// TwinCAT 3 PLC project DMMS_PLC
// ProgramVersion: 3.1.4026.19
// libraries:
//   Tc2_Standard, * (Beckhoff Automation GmbH)
//   Tc2_System, * (Beckhoff Automation GmbH)
//   Tc3_Mc3PlanarMotion, * (Beckhoff Automation GmbH)
//   Tc3_Physics, * (Beckhoff Automation GmbH)
//   Tc3_XPlanarStandard, * (Beckhoff Automation GmbH)
//   Tc3_XPlanarUtility, * (Beckhoff Automation GmbH)
// project tree:
//   DUTs/Communiction/GlobalStatus/ ST_ComIn_GlobalStatus.TcDUT (not stored), ST_ComOut_GlobalStatus.TcDUT (not stored), ST_Com_GlobalStatus.TcDUT (not stored)
//   DUTs/Communiction/Movers/ ST_ComIn_ExportMover.TcDUT (not stored), ST_ComOut_ExportMover.TcDUT, ST_Com_ExportMover.TcDUT (not stored)
//   DUTs/Communiction/Station/ ST_ComIn_ExportStation.TcDUT (not stored), ST_ComOut_ExportStation.TcDUT (not stored), ST_Com_ExportStation.TcDUT
//   GVLs/ Communication.TcGVL (not stored), Debug.TcGVL (not stored), GVL.TcGVL (not stored)
//   Mover/DUTs/ MoverPositionUnion.TcDUT, ST_ControlData.TcDUT (not stored), ST_EMoverLoadType.TcDUT (not stored), ST_ManMov_FreeMove.TcDUT, ST_ManMov_MoveTrack.TcDUT (not stored), ST_ManualMovements.TcDUT (not stored), ST_MoverConfiguration.TcDUT (not stored), ST_ProcessResult.TcDUT, ST_ProcessTask.TcDUT (not stored), ST_ProductData.TcDUT (not stored), ST_WellplateParametrization.TcDUT (not stored)
//   Mover/ FB_ApplicationMover.TcPOU, I_MoverApplication.TcIO
//   / PlcTask.TcTTO
//   POUs/ FB_MotionSystem.TcPOU, MAIN.TcPOU (not stored)
//   Stations/Base/ FB_StationBase.TcPOU, I_Station.TcIO
//   Stations/DUTs/ E_ProcessMode.TcDUT (not stored), ST_EStationProcessState.TcDUT (not stored), ST_EStationHandshake.TcDUT (not stored), ST_StationPosition.TcDUT (not stored), ST_StationReturn.TcDUT, ST_VisStationData.TcDUT (not stored)
//   Stations/ FB_PuncherStation.TcPOU (not stored), FB_PuncherSeparateStation.TcPOU, FB_PuncherBufferStation.TcPOU
//   Stations/Helper/ FB_HistoryInfo.TcPOU
//   Tracks/Base/ FB_BaseTrack.TcPOU (not stored), I_Track.TcIO (not stored)
//   Tracks/ FB_CloseLoopTrack.TcPOU (not stored), FB_UserInteractionTrack.TcPOU (not stored), FB_PipettePreBufferTrack.TcPOU (not stored), FB_PipetteTrack.TcPOU (not stored), FB_PipettePostBufferTrack.TcPOU, FB_PipetteBufferConTrack.TcPOU (not stored), FB_PuncherWellplateTrack.TcPOU, FB_PuncherBufferTrack.TcPOU (not stored), FB_StradeFirstSegTrack.TcPOU, FB_StradeSecondSegTrack.TcPOU (not stored), FB_PuncherSeperateTrack.TcPOU (not stored)
// real-time tasks:
//   TASK Job Task: cycle default, priority 2
//   TASK MC-Task (MET): cycle T#2ms, priority 3, ADS port 351
//   TASK MC-Task (MPT): cycle T#10ms, priority 4, ADS port 352
//   TASK PlcTask: cycle T#10ms, priority 20, ADS port 353
//   TASK XPlanar Task_0: cycle T#250us, priority 1, ADS port 350
//   TASK XPlanar Task_10: cycle T#250us, priority 5, ADS port 354
// I/O:
//   DEVICE Device 2 (EtherCAT), AmsNetId 192.168.2.44.3.1
//     Term 1 (APS4322-7000) [APS4322-7000 Drive]
//       Term 2 (APS4322-5000) [APS4322-5000 Feedback]
//     Term 3 (APS4322-7000) [APS4322-7000 Drive]
//       Term 4 (APS4322-5000) [APS4322-5000 Feedback]
//     Term 5 (APS4322-7000) [APS4322-7000 Drive]
//       Term 6 (APS4322-5000) [APS4322-5000 Feedback]
//     Term 7 (APS4322-7000) [APS4322-7000 Drive]
//       Term 8 (APS4322-5000) [APS4322-5000 Feedback]
//     Term 9 (APS4322-7000) [APS4322-7000 Drive]
//       Term 10 (APS4322-5000) [APS4322-5000 Feedback]
// variable links:
//   Device 2 (EtherCAT) <-> TcCOM Objects/XPlanar/Part1/APS4322_P1_1
//     Term 1 (APS4322-7000)/APS Comm Inputs/CommStatusWord <-> Data Pointer/MoverCommStatusWord
//     Term 1 (APS4322-7000)/APS Comm Inputs/Data {1..4} <-> Data Pointer/MoverCommDataIn[{0..3}]  (4 links)
//     Term 1 (APS4322-7000)/APS Comm Outputs/CommControlWord <-> Data Pointer/MoverCommControlWord
//     Term 1 (APS4322-7000)/APS Comm Outputs/Data 1 <-> Data Pointer/MoverCommDataOut
//     Term 1 (APS4322-7000)/APS Diagdata/DC Link Voltage <-> Data Pointer/DcLinkVoltage
//     Term 1 (APS4322-7000)/APS Diagdata/Power supply current <-> Data Pointer/PowerSupplyCurrent
//     Term 1 (APS4322-7000)/APS Inputs/StatusWord <-> Data Pointer/PowerUnitStatusWord
//     Term 1 (APS4322-7000)/APS Outputs/ControlWord <-> Data Pointer/PowerUnitControlWord
//     Term 1 (APS4322-7000)/APS Outputs/Current D 0X0 <-> Data Pointer/DCurrentSetPoints[0]
//     Term 1 (APS4322-7000)/APS Outputs/Current D 0X1 <-> Data Pointer/DCurrentSetPoints[1]
//     Term 1 (APS4322-7000)/APS Outputs/Current D 0X2 <-> Data Pointer/DCurrentSetPoints[2]
//     Term 1 (APS4322-7000)/APS Outputs/Current D 1X0 <-> Data Pointer/DCurrentSetPoints[6]
//     Term 1 (APS4322-7000)/APS Outputs/Current D 1X1 <-> Data Pointer/DCurrentSetPoints[7]
//     Term 1 (APS4322-7000)/APS Outputs/Current D 1X2 <-> Data Pointer/DCurrentSetPoints[8]
//     Term 1 (APS4322-7000)/APS Outputs/Current D 2X0 <-> Data Pointer/DCurrentSetPoints[12]
//     Term 1 (APS4322-7000)/APS Outputs/Current D 2X1 <-> Data Pointer/DCurrentSetPoints[13]
//     Term 1 (APS4322-7000)/APS Outputs/Current D 2X2 <-> Data Pointer/DCurrentSetPoints[14]
//     Term 1 (APS4322-7000)/APS Outputs/Current D 3X0 <-> Data Pointer/DCurrentSetPoints[18]
//     Term 1 (APS4322-7000)/APS Outputs/Current D 3X1 <-> Data Pointer/DCurrentSetPoints[19]
//     Term 1 (APS4322-7000)/APS Outputs/Current D 3X2 <-> Data Pointer/DCurrentSetPoints[20]
//     Term 1 (APS4322-7000)/APS Outputs/Current D 0Y0 <-> Data Pointer/DCurrentSetPoints[3]
//     Term 1 (APS4322-7000)/APS Outputs/Current D 0Y1 <-> Data Pointer/DCurrentSetPoints[4]
//     Term 1 (APS4322-7000)/APS Outputs/Current D 0Y2 <-> Data Pointer/DCurrentSetPoints[5]
//     Term 1 (APS4322-7000)/APS Outputs/Current D 1Y0 <-> Data Pointer/DCurrentSetPoints[9]
//     Term 1 (APS4322-7000)/APS Outputs/Current D 1Y1 <-> Data Pointer/DCurrentSetPoints[10]
//     Term 1 (APS4322-7000)/APS Outputs/Current D 1Y2 <-> Data Pointer/DCurrentSetPoints[11]
//     Term 1 (APS4322-7000)/APS Outputs/Current D 2Y0 <-> Data Pointer/DCurrentSetPoints[15]
//     Term 1 (APS4322-7000)/APS Outputs/Current D 2Y1 <-> Data Pointer/DCurrentSetPoints[16]
//     Term 1 (APS4322-7000)/APS Outputs/Current D 2Y2 <-> Data Pointer/DCurrentSetPoints[17]
//     Term 1 (APS4322-7000)/APS Outputs/Current D 3Y0 <-> Data Pointer/DCurrentSetPoints[21]
//     Term 1 (APS4322-7000)/APS Outputs/Current D 3Y1 <-> Data Pointer/DCurrentSetPoints[22]
//     Term 1 (APS4322-7000)/APS Outputs/Current D 3Y2 <-> Data Pointer/DCurrentSetPoints[23]
//     Term 1 (APS4322-7000)/APS Outputs/Current Q 0X0 <-> Data Pointer/QCurrentSetPoints[0]
//     Term 1 (APS4322-7000)/APS Outputs/Current Q 0X1 <-> Data Pointer/QCurrentSetPoints[1]
//     Term 1 (APS4322-7000)/APS Outputs/Current Q 0X2 <-> Data Pointer/QCurrentSetPoints[2]
//     Term 1 (APS4322-7000)/APS Outputs/Current Q 1X0 <-> Data Pointer/QCurrentSetPoints[6]
//     Term 1 (APS4322-7000)/APS Outputs/Current Q 1X1 <-> Data Pointer/QCurrentSetPoints[7]
//     Term 1 (APS4322-7000)/APS Outputs/Current Q 1X2 <-> Data Pointer/QCurrentSetPoints[8]
//     Term 1 (APS4322-7000)/APS Outputs/Current Q 2X0 <-> Data Pointer/QCurrentSetPoints[12]
//     Term 1 (APS4322-7000)/APS Outputs/Current Q 2X1 <-> Data Pointer/QCurrentSetPoints[13]
//     Term 1 (APS4322-7000)/APS Outputs/Current Q 2X2 <-> Data Pointer/QCurrentSetPoints[14]
//     Term 1 (APS4322-7000)/APS Outputs/Current Q 3X0 <-> Data Pointer/QCurrentSetPoints[18]
//     Term 1 (APS4322-7000)/APS Outputs/Current Q 3X1 <-> Data Pointer/QCurrentSetPoints[19]
//     Term 1 (APS4322-7000)/APS Outputs/Current Q 3X2 <-> Data Pointer/QCurrentSetPoints[20]
//     Term 1 (APS4322-7000)/APS Outputs/Current Q 0Y0 <-> Data Pointer/QCurrentSetPoints[3]
//     Term 1 (APS4322-7000)/APS Outputs/Current Q 0Y1 <-> Data Pointer/QCurrentSetPoints[4]
//     Term 1 (APS4322-7000)/APS Outputs/Current Q 0Y2 <-> Data Pointer/QCurrentSetPoints[5]
//     Term 1 (APS4322-7000)/APS Outputs/Current Q 1Y0 <-> Data Pointer/QCurrentSetPoints[9]
//     Term 1 (APS4322-7000)/APS Outputs/Current Q 1Y1 <-> Data Pointer/QCurrentSetPoints[10]
//     Term 1 (APS4322-7000)/APS Outputs/Current Q 1Y2 <-> Data Pointer/QCurrentSetPoints[11]
//     Term 1 (APS4322-7000)/APS Outputs/Current Q 2Y0 <-> Data Pointer/QCurrentSetPoints[15]
//     Term 1 (APS4322-7000)/APS Outputs/Current Q 2Y1 <-> Data Pointer/QCurrentSetPoints[16]
//     Term 1 (APS4322-7000)/APS Outputs/Current Q 2Y2 <-> Data Pointer/QCurrentSetPoints[17]
//     Term 1 (APS4322-7000)/APS Outputs/Current Q 3Y0 <-> Data Pointer/QCurrentSetPoints[21]
//     Term 1 (APS4322-7000)/APS Outputs/Current Q 3Y1 <-> Data Pointer/QCurrentSetPoints[22]
//     Term 1 (APS4322-7000)/APS Outputs/Current Q 3Y2 <-> Data Pointer/QCurrentSetPoints[23]
//     Term 1 (APS4322-7000)/APS Outputs/PhiE 0X0 <-> Data Pointer/PhiSetPoints[0]
//     Term 1 (APS4322-7000)/APS Outputs/PhiE 0X1 <-> Data Pointer/PhiSetPoints[1]
//     Term 1 (APS4322-7000)/APS Outputs/PhiE 0X2 <-> Data Pointer/PhiSetPoints[2]
//     Term 1 (APS4322-7000)/APS Outputs/PhiE 1X0 <-> Data Pointer/PhiSetPoints[6]
//     Term 1 (APS4322-7000)/APS Outputs/PhiE 1X1 <-> Data Pointer/PhiSetPoints[7]
//     Term 1 (APS4322-7000)/APS Outputs/PhiE 1X2 <-> Data Pointer/PhiSetPoints[8]
//     Term 1 (APS4322-7000)/APS Outputs/PhiE 2X0 <-> Data Pointer/PhiSetPoints[12]
//     Term 1 (APS4322-7000)/APS Outputs/PhiE 2X1 <-> Data Pointer/PhiSetPoints[13]
//     Term 1 (APS4322-7000)/APS Outputs/PhiE 2X2 <-> Data Pointer/PhiSetPoints[14]
//     Term 1 (APS4322-7000)/APS Outputs/PhiE 3X0 <-> Data Pointer/PhiSetPoints[18]
//     Term 1 (APS4322-7000)/APS Outputs/PhiE 3X1 <-> Data Pointer/PhiSetPoints[19]
//     Term 1 (APS4322-7000)/APS Outputs/PhiE 3X2 <-> Data Pointer/PhiSetPoints[20]
//     Term 1 (APS4322-7000)/APS Outputs/PhiE 0Y0 <-> Data Pointer/PhiSetPoints[3]
//     Term 1 (APS4322-7000)/APS Outputs/PhiE 0Y1 <-> Data Pointer/PhiSetPoints[4]
//     Term 1 (APS4322-7000)/APS Outputs/PhiE 0Y2 <-> Data Pointer/PhiSetPoints[5]
//     Term 1 (APS4322-7000)/APS Outputs/PhiE 1Y0 <-> Data Pointer/PhiSetPoints[9]
//     Term 1 (APS4322-7000)/APS Outputs/PhiE 1Y1 <-> Data Pointer/PhiSetPoints[10]
//     Term 1 (APS4322-7000)/APS Outputs/PhiE 1Y2 <-> Data Pointer/PhiSetPoints[11]
//     Term 1 (APS4322-7000)/APS Outputs/PhiE 2Y0 <-> Data Pointer/PhiSetPoints[15]
//     Term 1 (APS4322-7000)/APS Outputs/PhiE 2Y1 <-> Data Pointer/PhiSetPoints[16]
//     Term 1 (APS4322-7000)/APS Outputs/PhiE 2Y2 <-> Data Pointer/PhiSetPoints[17]
//     Term 1 (APS4322-7000)/APS Outputs/PhiE 3Y0 <-> Data Pointer/PhiSetPoints[21]
//     Term 1 (APS4322-7000)/APS Outputs/PhiE 3Y1 <-> Data Pointer/PhiSetPoints[22]
//     Term 1 (APS4322-7000)/APS Outputs/PhiE 3Y2 <-> Data Pointer/PhiSetPoints[23]
//     Term 1 (APS4322-7000)/Term 2 (APS4322-5000)/FB Inputs/A{0..8 step 2} X-Field <-> Data Pointer/HallSensorFieldsXYZ[{0..12 step 3}]  (5 links)
//     Term 1 (APS4322-7000)/Term 2 (APS4322-5000)/FB Inputs/A{0..8 step 2} Y-Field <-> Data Pointer/HallSensorFieldsXYZ[{1..13 step 3}]  (5 links)
//     Term 1 (APS4322-7000)/Term 2 (APS4322-5000)/FB Inputs/A{0..8 step 2} Z-Field <-> Data Pointer/HallSensorFieldsXYZ[{2..14 step 3}]  (5 links)
//     Term 1 (APS4322-7000)/Term 2 (APS4322-5000)/FB Inputs/B{1..9 step 2} X-Field <-> Data Pointer/HallSensorFieldsXYZ[{15..27 step 3}]  (5 links)
//     Term 1 (APS4322-7000)/Term 2 (APS4322-5000)/FB Inputs/B{1..9 step 2} Y-Field <-> Data Pointer/HallSensorFieldsXYZ[{16..28 step 3}]  (5 links)
//     Term 1 (APS4322-7000)/Term 2 (APS4322-5000)/FB Inputs/B{1..9 step 2} Z-Field <-> Data Pointer/HallSensorFieldsXYZ[{17..29 step 3}]  (5 links)
//     Term 1 (APS4322-7000)/Term 2 (APS4322-5000)/FB Inputs/C{0..8 step 2} X-Field <-> Data Pointer/HallSensorFieldsXYZ[{30..42 step 3}]  (5 links)
//     Term 1 (APS4322-7000)/Term 2 (APS4322-5000)/FB Inputs/C{0..8 step 2} Y-Field <-> Data Pointer/HallSensorFieldsXYZ[{31..43 step 3}]  (5 links)
//     Term 1 (APS4322-7000)/Term 2 (APS4322-5000)/FB Inputs/C{0..8 step 2} Z-Field <-> Data Pointer/HallSensorFieldsXYZ[{32..44 step 3}]  (5 links)
//     Term 1 (APS4322-7000)/Term 2 (APS4322-5000)/FB Inputs/D{1..9 step 2} X-Field <-> Data Pointer/HallSensorFieldsXYZ[{45..57 step 3}]  (5 links)
//     Term 1 (APS4322-7000)/Term 2 (APS4322-5000)/FB Inputs/D{1..9 step 2} Y-Field <-> Data Pointer/HallSensorFieldsXYZ[{46..58 step 3}]  (5 links)
//     Term 1 (APS4322-7000)/Term 2 (APS4322-5000)/FB Inputs/D{1..9 step 2} Z-Field <-> Data Pointer/HallSensorFieldsXYZ[{47..59 step 3}]  (5 links)
//     Term 1 (APS4322-7000)/Term 2 (APS4322-5000)/FB Inputs/E{0..8 step 2} X-Field <-> Data Pointer/HallSensorFieldsXYZ[{60..72 step 3}]  (5 links)
//     Term 1 (APS4322-7000)/Term 2 (APS4322-5000)/FB Inputs/E{0..8 step 2} Y-Field <-> Data Pointer/HallSensorFieldsXYZ[{61..73 step 3}]  (5 links)
//     Term 1 (APS4322-7000)/Term 2 (APS4322-5000)/FB Inputs/E{0..8 step 2} Z-Field <-> Data Pointer/HallSensorFieldsXYZ[{62..74 step 3}]  (5 links)
//     Term 1 (APS4322-7000)/Term 2 (APS4322-5000)/FB Inputs/F{1..9 step 2} X-Field <-> Data Pointer/HallSensorFieldsXYZ[{75..87 step 3}]  (5 links)
//     Term 1 (APS4322-7000)/Term 2 (APS4322-5000)/FB Inputs/F{1..9 step 2} Y-Field <-> Data Pointer/HallSensorFieldsXYZ[{76..88 step 3}]  (5 links)
//     Term 1 (APS4322-7000)/Term 2 (APS4322-5000)/FB Inputs/F{1..9 step 2} Z-Field <-> Data Pointer/HallSensorFieldsXYZ[{77..89 step 3}]  (5 links)
//     Term 1 (APS4322-7000)/Term 2 (APS4322-5000)/FB Inputs/G{0..8 step 2} X-Field <-> Data Pointer/HallSensorFieldsXYZ[{90..102 step 3}]  (5 links)
//     Term 1 (APS4322-7000)/Term 2 (APS4322-5000)/FB Inputs/G{0..8 step 2} Y-Field <-> Data Pointer/HallSensorFieldsXYZ[{91..103 step 3}]  (5 links)
//     Term 1 (APS4322-7000)/Term 2 (APS4322-5000)/FB Inputs/G{0..8 step 2} Z-Field <-> Data Pointer/HallSensorFieldsXYZ[{92..104 step 3}]  (5 links)
//     Term 1 (APS4322-7000)/Term 2 (APS4322-5000)/FB Inputs/H{1..9 step 2} X-Field <-> Data Pointer/HallSensorFieldsXYZ[{105..117 step 3}]  (5 links)
//     Term 1 (APS4322-7000)/Term 2 (APS4322-5000)/FB Inputs/H{1..9 step 2} Y-Field <-> Data Pointer/HallSensorFieldsXYZ[{106..118 step 3}]  (5 links)
//     Term 1 (APS4322-7000)/Term 2 (APS4322-5000)/FB Inputs/H{1..9 step 2} Z-Field <-> Data Pointer/HallSensorFieldsXYZ[{107..119 step 3}]  (5 links)
//     Term 1 (APS4322-7000)/Term 2 (APS4322-5000)/FB Inputs/I{0..8 step 2} X-Field <-> Data Pointer/HallSensorFieldsXYZ[{120..132 step 3}]  (5 links)
//     Term 1 (APS4322-7000)/Term 2 (APS4322-5000)/FB Inputs/I{0..8 step 2} Y-Field <-> Data Pointer/HallSensorFieldsXYZ[{121..133 step 3}]  (5 links)
//     Term 1 (APS4322-7000)/Term 2 (APS4322-5000)/FB Inputs/I{0..8 step 2} Z-Field <-> Data Pointer/HallSensorFieldsXYZ[{122..134 step 3}]  (5 links)
//     Term 1 (APS4322-7000)/Term 2 (APS4322-5000)/FB Inputs/J{1..9 step 2} X-Field <-> Data Pointer/HallSensorFieldsXYZ[{135..147 step 3}]  (5 links)
//     Term 1 (APS4322-7000)/Term 2 (APS4322-5000)/FB Inputs/J{1..9 step 2} Y-Field <-> Data Pointer/HallSensorFieldsXYZ[{136..148 step 3}]  (5 links)
//     Term 1 (APS4322-7000)/Term 2 (APS4322-5000)/FB Inputs/J{1..9 step 2} Z-Field <-> Data Pointer/HallSensorFieldsXYZ[{137..149 step 3}]  (5 links)
//     Term 1 (APS4322-7000)/Term 2 (APS4322-5000)/FB Inputs/Status <-> Data Pointer/FeedbackStatus
//   Device 2 (EtherCAT) <-> TcCOM Objects/XPlanar/Part1/APS4322_P1_2
//     Term 3 (APS4322-7000)/APS Comm Inputs/CommStatusWord <-> Data Pointer/MoverCommStatusWord
//     Term 3 (APS4322-7000)/APS Comm Inputs/Data {1..4} <-> Data Pointer/MoverCommDataIn[{0..3}]  (4 links)
//     Term 3 (APS4322-7000)/APS Comm Outputs/CommControlWord <-> Data Pointer/MoverCommControlWord
//     Term 3 (APS4322-7000)/APS Comm Outputs/Data 1 <-> Data Pointer/MoverCommDataOut
//     Term 3 (APS4322-7000)/APS Diagdata/DC Link Voltage <-> Data Pointer/DcLinkVoltage
//     Term 3 (APS4322-7000)/APS Diagdata/Power supply current <-> Data Pointer/PowerSupplyCurrent
//     Term 3 (APS4322-7000)/APS Inputs/StatusWord <-> Data Pointer/PowerUnitStatusWord
//     Term 3 (APS4322-7000)/APS Outputs/ControlWord <-> Data Pointer/PowerUnitControlWord
//     Term 3 (APS4322-7000)/APS Outputs/Current D 0X0 <-> Data Pointer/DCurrentSetPoints[0]
//     Term 3 (APS4322-7000)/APS Outputs/Current D 0X1 <-> Data Pointer/DCurrentSetPoints[1]
//     Term 3 (APS4322-7000)/APS Outputs/Current D 0X2 <-> Data Pointer/DCurrentSetPoints[2]
//     Term 3 (APS4322-7000)/APS Outputs/Current D 1X0 <-> Data Pointer/DCurrentSetPoints[6]
//     Term 3 (APS4322-7000)/APS Outputs/Current D 1X1 <-> Data Pointer/DCurrentSetPoints[7]
//     Term 3 (APS4322-7000)/APS Outputs/Current D 1X2 <-> Data Pointer/DCurrentSetPoints[8]
//     Term 3 (APS4322-7000)/APS Outputs/Current D 2X0 <-> Data Pointer/DCurrentSetPoints[12]
//     Term 3 (APS4322-7000)/APS Outputs/Current D 2X1 <-> Data Pointer/DCurrentSetPoints[13]
//     Term 3 (APS4322-7000)/APS Outputs/Current D 2X2 <-> Data Pointer/DCurrentSetPoints[14]
//     Term 3 (APS4322-7000)/APS Outputs/Current D 3X0 <-> Data Pointer/DCurrentSetPoints[18]
//     Term 3 (APS4322-7000)/APS Outputs/Current D 3X1 <-> Data Pointer/DCurrentSetPoints[19]
//     Term 3 (APS4322-7000)/APS Outputs/Current D 3X2 <-> Data Pointer/DCurrentSetPoints[20]
//     Term 3 (APS4322-7000)/APS Outputs/Current D 0Y0 <-> Data Pointer/DCurrentSetPoints[3]
//     Term 3 (APS4322-7000)/APS Outputs/Current D 0Y1 <-> Data Pointer/DCurrentSetPoints[4]
//     Term 3 (APS4322-7000)/APS Outputs/Current D 0Y2 <-> Data Pointer/DCurrentSetPoints[5]
//     Term 3 (APS4322-7000)/APS Outputs/Current D 1Y0 <-> Data Pointer/DCurrentSetPoints[9]
//     Term 3 (APS4322-7000)/APS Outputs/Current D 1Y1 <-> Data Pointer/DCurrentSetPoints[10]
//     Term 3 (APS4322-7000)/APS Outputs/Current D 1Y2 <-> Data Pointer/DCurrentSetPoints[11]
//     Term 3 (APS4322-7000)/APS Outputs/Current D 2Y0 <-> Data Pointer/DCurrentSetPoints[15]
//     Term 3 (APS4322-7000)/APS Outputs/Current D 2Y1 <-> Data Pointer/DCurrentSetPoints[16]
//     Term 3 (APS4322-7000)/APS Outputs/Current D 2Y2 <-> Data Pointer/DCurrentSetPoints[17]
//     Term 3 (APS4322-7000)/APS Outputs/Current D 3Y0 <-> Data Pointer/DCurrentSetPoints[21]
//     Term 3 (APS4322-7000)/APS Outputs/Current D 3Y1 <-> Data Pointer/DCurrentSetPoints[22]
//     Term 3 (APS4322-7000)/APS Outputs/Current D 3Y2 <-> Data Pointer/DCurrentSetPoints[23]
//     Term 3 (APS4322-7000)/APS Outputs/Current Q 0X0 <-> Data Pointer/QCurrentSetPoints[0]
//     Term 3 (APS4322-7000)/APS Outputs/Current Q 0X1 <-> Data Pointer/QCurrentSetPoints[1]
//     Term 3 (APS4322-7000)/APS Outputs/Current Q 0X2 <-> Data Pointer/QCurrentSetPoints[2]
//     Term 3 (APS4322-7000)/APS Outputs/Current Q 1X0 <-> Data Pointer/QCurrentSetPoints[6]
//     Term 3 (APS4322-7000)/APS Outputs/Current Q 1X1 <-> Data Pointer/QCurrentSetPoints[7]
//     Term 3 (APS4322-7000)/APS Outputs/Current Q 1X2 <-> Data Pointer/QCurrentSetPoints[8]
//     Term 3 (APS4322-7000)/APS Outputs/Current Q 2X0 <-> Data Pointer/QCurrentSetPoints[12]
//     Term 3 (APS4322-7000)/APS Outputs/Current Q 2X1 <-> Data Pointer/QCurrentSetPoints[13]
//     Term 3 (APS4322-7000)/APS Outputs/Current Q 2X2 <-> Data Pointer/QCurrentSetPoints[14]
//     Term 3 (APS4322-7000)/APS Outputs/Current Q 3X0 <-> Data Pointer/QCurrentSetPoints[18]
//     Term 3 (APS4322-7000)/APS Outputs/Current Q 3X1 <-> Data Pointer/QCurrentSetPoints[19]
//     Term 3 (APS4322-7000)/APS Outputs/Current Q 3X2 <-> Data Pointer/QCurrentSetPoints[20]
//     Term 3 (APS4322-7000)/APS Outputs/Current Q 0Y0 <-> Data Pointer/QCurrentSetPoints[3]
//     Term 3 (APS4322-7000)/APS Outputs/Current Q 0Y1 <-> Data Pointer/QCurrentSetPoints[4]
//     Term 3 (APS4322-7000)/APS Outputs/Current Q 0Y2 <-> Data Pointer/QCurrentSetPoints[5]
//     Term 3 (APS4322-7000)/APS Outputs/Current Q 1Y0 <-> Data Pointer/QCurrentSetPoints[9]
//     Term 3 (APS4322-7000)/APS Outputs/Current Q 1Y1 <-> Data Pointer/QCurrentSetPoints[10]
//     Term 3 (APS4322-7000)/APS Outputs/Current Q 1Y2 <-> Data Pointer/QCurrentSetPoints[11]
//     Term 3 (APS4322-7000)/APS Outputs/Current Q 2Y0 <-> Data Pointer/QCurrentSetPoints[15]
//     Term 3 (APS4322-7000)/APS Outputs/Current Q 2Y1 <-> Data Pointer/QCurrentSetPoints[16]
//     Term 3 (APS4322-7000)/APS Outputs/Current Q 2Y2 <-> Data Pointer/QCurrentSetPoints[17]
//     Term 3 (APS4322-7000)/APS Outputs/Current Q 3Y0 <-> Data Pointer/QCurrentSetPoints[21]
//     Term 3 (APS4322-7000)/APS Outputs/Current Q 3Y1 <-> Data Pointer/QCurrentSetPoints[22]
//     Term 3 (APS4322-7000)/APS Outputs/Current Q 3Y2 <-> Data Pointer/QCurrentSetPoints[23]
//     Term 3 (APS4322-7000)/APS Outputs/PhiE 0X0 <-> Data Pointer/PhiSetPoints[0]
//     Term 3 (APS4322-7000)/APS Outputs/PhiE 0X1 <-> Data Pointer/PhiSetPoints[1]
//     Term 3 (APS4322-7000)/APS Outputs/PhiE 0X2 <-> Data Pointer/PhiSetPoints[2]
//     Term 3 (APS4322-7000)/APS Outputs/PhiE 1X0 <-> Data Pointer/PhiSetPoints[6]
//     Term 3 (APS4322-7000)/APS Outputs/PhiE 1X1 <-> Data Pointer/PhiSetPoints[7]
//     Term 3 (APS4322-7000)/APS Outputs/PhiE 1X2 <-> Data Pointer/PhiSetPoints[8]
//     Term 3 (APS4322-7000)/APS Outputs/PhiE 2X0 <-> Data Pointer/PhiSetPoints[12]
//     Term 3 (APS4322-7000)/APS Outputs/PhiE 2X1 <-> Data Pointer/PhiSetPoints[13]
//     Term 3 (APS4322-7000)/APS Outputs/PhiE 2X2 <-> Data Pointer/PhiSetPoints[14]
//     Term 3 (APS4322-7000)/APS Outputs/PhiE 3X0 <-> Data Pointer/PhiSetPoints[18]
//     Term 3 (APS4322-7000)/APS Outputs/PhiE 3X1 <-> Data Pointer/PhiSetPoints[19]
//     Term 3 (APS4322-7000)/APS Outputs/PhiE 3X2 <-> Data Pointer/PhiSetPoints[20]
//     Term 3 (APS4322-7000)/APS Outputs/PhiE 0Y0 <-> Data Pointer/PhiSetPoints[3]
//     Term 3 (APS4322-7000)/APS Outputs/PhiE 0Y1 <-> Data Pointer/PhiSetPoints[4]
//     Term 3 (APS4322-7000)/APS Outputs/PhiE 0Y2 <-> Data Pointer/PhiSetPoints[5]
//     Term 3 (APS4322-7000)/APS Outputs/PhiE 1Y0 <-> Data Pointer/PhiSetPoints[9]
//     Term 3 (APS4322-7000)/APS Outputs/PhiE 1Y1 <-> Data Pointer/PhiSetPoints[10]
//     Term 3 (APS4322-7000)/APS Outputs/PhiE 1Y2 <-> Data Pointer/PhiSetPoints[11]
//     Term 3 (APS4322-7000)/APS Outputs/PhiE 2Y0 <-> Data Pointer/PhiSetPoints[15]
//     Term 3 (APS4322-7000)/APS Outputs/PhiE 2Y1 <-> Data Pointer/PhiSetPoints[16]
//     Term 3 (APS4322-7000)/APS Outputs/PhiE 2Y2 <-> Data Pointer/PhiSetPoints[17]
//     Term 3 (APS4322-7000)/APS Outputs/PhiE 3Y0 <-> Data Pointer/PhiSetPoints[21]
//     Term 3 (APS4322-7000)/APS Outputs/PhiE 3Y1 <-> Data Pointer/PhiSetPoints[22]
//     Term 3 (APS4322-7000)/APS Outputs/PhiE 3Y2 <-> Data Pointer/PhiSetPoints[23]
//     Term 3 (APS4322-7000)/Term 4 (APS4322-5000)/FB Inputs/A{0..8 step 2} X-Field <-> Data Pointer/HallSensorFieldsXYZ[{0..12 step 3}]  (5 links)
//     Term 3 (APS4322-7000)/Term 4 (APS4322-5000)/FB Inputs/A{0..8 step 2} Y-Field <-> Data Pointer/HallSensorFieldsXYZ[{1..13 step 3}]  (5 links)
//     Term 3 (APS4322-7000)/Term 4 (APS4322-5000)/FB Inputs/A{0..8 step 2} Z-Field <-> Data Pointer/HallSensorFieldsXYZ[{2..14 step 3}]  (5 links)
//     Term 3 (APS4322-7000)/Term 4 (APS4322-5000)/FB Inputs/B{1..9 step 2} X-Field <-> Data Pointer/HallSensorFieldsXYZ[{15..27 step 3}]  (5 links)
//     Term 3 (APS4322-7000)/Term 4 (APS4322-5000)/FB Inputs/B{1..9 step 2} Y-Field <-> Data Pointer/HallSensorFieldsXYZ[{16..28 step 3}]  (5 links)
//     Term 3 (APS4322-7000)/Term 4 (APS4322-5000)/FB Inputs/B{1..9 step 2} Z-Field <-> Data Pointer/HallSensorFieldsXYZ[{17..29 step 3}]  (5 links)
//     Term 3 (APS4322-7000)/Term 4 (APS4322-5000)/FB Inputs/C{0..8 step 2} X-Field <-> Data Pointer/HallSensorFieldsXYZ[{30..42 step 3}]  (5 links)
//     Term 3 (APS4322-7000)/Term 4 (APS4322-5000)/FB Inputs/C{0..8 step 2} Y-Field <-> Data Pointer/HallSensorFieldsXYZ[{31..43 step 3}]  (5 links)
//     Term 3 (APS4322-7000)/Term 4 (APS4322-5000)/FB Inputs/C{0..8 step 2} Z-Field <-> Data Pointer/HallSensorFieldsXYZ[{32..44 step 3}]  (5 links)
//     Term 3 (APS4322-7000)/Term 4 (APS4322-5000)/FB Inputs/D{1..9 step 2} X-Field <-> Data Pointer/HallSensorFieldsXYZ[{45..57 step 3}]  (5 links)
//     Term 3 (APS4322-7000)/Term 4 (APS4322-5000)/FB Inputs/D{1..9 step 2} Y-Field <-> Data Pointer/HallSensorFieldsXYZ[{46..58 step 3}]  (5 links)
//     Term 3 (APS4322-7000)/Term 4 (APS4322-5000)/FB Inputs/D{1..9 step 2} Z-Field <-> Data Pointer/HallSensorFieldsXYZ[{47..59 step 3}]  (5 links)
//     Term 3 (APS4322-7000)/Term 4 (APS4322-5000)/FB Inputs/E{0..8 step 2} X-Field <-> Data Pointer/HallSensorFieldsXYZ[{60..72 step 3}]  (5 links)
//     Term 3 (APS4322-7000)/Term 4 (APS4322-5000)/FB Inputs/E{0..8 step 2} Y-Field <-> Data Pointer/HallSensorFieldsXYZ[{61..73 step 3}]  (5 links)
//     Term 3 (APS4322-7000)/Term 4 (APS4322-5000)/FB Inputs/E{0..8 step 2} Z-Field <-> Data Pointer/HallSensorFieldsXYZ[{62..74 step 3}]  (5 links)
//     Term 3 (APS4322-7000)/Term 4 (APS4322-5000)/FB Inputs/F{1..9 step 2} X-Field <-> Data Pointer/HallSensorFieldsXYZ[{75..87 step 3}]  (5 links)
//     Term 3 (APS4322-7000)/Term 4 (APS4322-5000)/FB Inputs/F{1..9 step 2} Y-Field <-> Data Pointer/HallSensorFieldsXYZ[{76..88 step 3}]  (5 links)
//     Term 3 (APS4322-7000)/Term 4 (APS4322-5000)/FB Inputs/F{1..9 step 2} Z-Field <-> Data Pointer/HallSensorFieldsXYZ[{77..89 step 3}]  (5 links)
//     Term 3 (APS4322-7000)/Term 4 (APS4322-5000)/FB Inputs/G{0..8 step 2} X-Field <-> Data Pointer/HallSensorFieldsXYZ[{90..102 step 3}]  (5 links)
//     Term 3 (APS4322-7000)/Term 4 (APS4322-5000)/FB Inputs/G{0..8 step 2} Y-Field <-> Data Pointer/HallSensorFieldsXYZ[{91..103 step 3}]  (5 links)
//     Term 3 (APS4322-7000)/Term 4 (APS4322-5000)/FB Inputs/G{0..8 step 2} Z-Field <-> Data Pointer/HallSensorFieldsXYZ[{92..104 step 3}]  (5 links)
//     Term 3 (APS4322-7000)/Term 4 (APS4322-5000)/FB Inputs/H{1..9 step 2} X-Field <-> Data Pointer/HallSensorFieldsXYZ[{105..117 step 3}]  (5 links)
//     Term 3 (APS4322-7000)/Term 4 (APS4322-5000)/FB Inputs/H{1..9 step 2} Y-Field <-> Data Pointer/HallSensorFieldsXYZ[{106..118 step 3}]  (5 links)
//     Term 3 (APS4322-7000)/Term 4 (APS4322-5000)/FB Inputs/H{1..9 step 2} Z-Field <-> Data Pointer/HallSensorFieldsXYZ[{107..119 step 3}]  (5 links)
//     Term 3 (APS4322-7000)/Term 4 (APS4322-5000)/FB Inputs/I{0..8 step 2} X-Field <-> Data Pointer/HallSensorFieldsXYZ[{120..132 step 3}]  (5 links)
//     Term 3 (APS4322-7000)/Term 4 (APS4322-5000)/FB Inputs/I{0..8 step 2} Y-Field <-> Data Pointer/HallSensorFieldsXYZ[{121..133 step 3}]  (5 links)
//     Term 3 (APS4322-7000)/Term 4 (APS4322-5000)/FB Inputs/I{0..8 step 2} Z-Field <-> Data Pointer/HallSensorFieldsXYZ[{122..134 step 3}]  (5 links)
//     Term 3 (APS4322-7000)/Term 4 (APS4322-5000)/FB Inputs/J{1..9 step 2} X-Field <-> Data Pointer/HallSensorFieldsXYZ[{135..147 step 3}]  (5 links)
//     Term 3 (APS4322-7000)/Term 4 (APS4322-5000)/FB Inputs/J{1..9 step 2} Y-Field <-> Data Pointer/HallSensorFieldsXYZ[{136..148 step 3}]  (5 links)
//     Term 3 (APS4322-7000)/Term 4 (APS4322-5000)/FB Inputs/J{1..9 step 2} Z-Field <-> Data Pointer/HallSensorFieldsXYZ[{137..149 step 3}]  (5 links)
//     Term 3 (APS4322-7000)/Term 4 (APS4322-5000)/FB Inputs/Status <-> Data Pointer/FeedbackStatus
//   Device 2 (EtherCAT) <-> TcCOM Objects/XPlanar/Part1/APS4322_P1_3
//     Term 5 (APS4322-7000)/APS Comm Inputs/CommStatusWord <-> Data Pointer/MoverCommStatusWord
//     Term 5 (APS4322-7000)/APS Comm Inputs/Data {1..4} <-> Data Pointer/MoverCommDataIn[{0..3}]  (4 links)
//     Term 5 (APS4322-7000)/APS Comm Outputs/CommControlWord <-> Data Pointer/MoverCommControlWord
//     Term 5 (APS4322-7000)/APS Comm Outputs/Data 1 <-> Data Pointer/MoverCommDataOut
//     Term 5 (APS4322-7000)/APS Diagdata/DC Link Voltage <-> Data Pointer/DcLinkVoltage
//     Term 5 (APS4322-7000)/APS Diagdata/Power supply current <-> Data Pointer/PowerSupplyCurrent
//     Term 5 (APS4322-7000)/APS Inputs/StatusWord <-> Data Pointer/PowerUnitStatusWord
//     Term 5 (APS4322-7000)/APS Outputs/ControlWord <-> Data Pointer/PowerUnitControlWord
//     Term 5 (APS4322-7000)/APS Outputs/Current D 0X0 <-> Data Pointer/DCurrentSetPoints[0]
//     Term 5 (APS4322-7000)/APS Outputs/Current D 0X1 <-> Data Pointer/DCurrentSetPoints[1]
//     Term 5 (APS4322-7000)/APS Outputs/Current D 0X2 <-> Data Pointer/DCurrentSetPoints[2]
//     Term 5 (APS4322-7000)/APS Outputs/Current D 1X0 <-> Data Pointer/DCurrentSetPoints[6]
//     Term 5 (APS4322-7000)/APS Outputs/Current D 1X1 <-> Data Pointer/DCurrentSetPoints[7]
//     Term 5 (APS4322-7000)/APS Outputs/Current D 1X2 <-> Data Pointer/DCurrentSetPoints[8]
//     Term 5 (APS4322-7000)/APS Outputs/Current D 2X0 <-> Data Pointer/DCurrentSetPoints[12]
//     Term 5 (APS4322-7000)/APS Outputs/Current D 2X1 <-> Data Pointer/DCurrentSetPoints[13]
//     Term 5 (APS4322-7000)/APS Outputs/Current D 2X2 <-> Data Pointer/DCurrentSetPoints[14]
//     Term 5 (APS4322-7000)/APS Outputs/Current D 3X0 <-> Data Pointer/DCurrentSetPoints[18]
//     Term 5 (APS4322-7000)/APS Outputs/Current D 3X1 <-> Data Pointer/DCurrentSetPoints[19]
//     Term 5 (APS4322-7000)/APS Outputs/Current D 3X2 <-> Data Pointer/DCurrentSetPoints[20]
//     Term 5 (APS4322-7000)/APS Outputs/Current D 0Y0 <-> Data Pointer/DCurrentSetPoints[3]
//     Term 5 (APS4322-7000)/APS Outputs/Current D 0Y1 <-> Data Pointer/DCurrentSetPoints[4]
//     Term 5 (APS4322-7000)/APS Outputs/Current D 0Y2 <-> Data Pointer/DCurrentSetPoints[5]
//     Term 5 (APS4322-7000)/APS Outputs/Current D 1Y0 <-> Data Pointer/DCurrentSetPoints[9]
//     Term 5 (APS4322-7000)/APS Outputs/Current D 1Y1 <-> Data Pointer/DCurrentSetPoints[10]
//     Term 5 (APS4322-7000)/APS Outputs/Current D 1Y2 <-> Data Pointer/DCurrentSetPoints[11]
//     Term 5 (APS4322-7000)/APS Outputs/Current D 2Y0 <-> Data Pointer/DCurrentSetPoints[15]
//     Term 5 (APS4322-7000)/APS Outputs/Current D 2Y1 <-> Data Pointer/DCurrentSetPoints[16]
//     Term 5 (APS4322-7000)/APS Outputs/Current D 2Y2 <-> Data Pointer/DCurrentSetPoints[17]
//     Term 5 (APS4322-7000)/APS Outputs/Current D 3Y0 <-> Data Pointer/DCurrentSetPoints[21]
//     Term 5 (APS4322-7000)/APS Outputs/Current D 3Y1 <-> Data Pointer/DCurrentSetPoints[22]
//     Term 5 (APS4322-7000)/APS Outputs/Current D 3Y2 <-> Data Pointer/DCurrentSetPoints[23]
//     Term 5 (APS4322-7000)/APS Outputs/Current Q 0X0 <-> Data Pointer/QCurrentSetPoints[0]
//     Term 5 (APS4322-7000)/APS Outputs/Current Q 0X1 <-> Data Pointer/QCurrentSetPoints[1]
//     Term 5 (APS4322-7000)/APS Outputs/Current Q 0X2 <-> Data Pointer/QCurrentSetPoints[2]
//     Term 5 (APS4322-7000)/APS Outputs/Current Q 1X0 <-> Data Pointer/QCurrentSetPoints[6]
//     Term 5 (APS4322-7000)/APS Outputs/Current Q 1X1 <-> Data Pointer/QCurrentSetPoints[7]
//     Term 5 (APS4322-7000)/APS Outputs/Current Q 1X2 <-> Data Pointer/QCurrentSetPoints[8]
//     Term 5 (APS4322-7000)/APS Outputs/Current Q 2X0 <-> Data Pointer/QCurrentSetPoints[12]
//     Term 5 (APS4322-7000)/APS Outputs/Current Q 2X1 <-> Data Pointer/QCurrentSetPoints[13]
//     Term 5 (APS4322-7000)/APS Outputs/Current Q 2X2 <-> Data Pointer/QCurrentSetPoints[14]
//     Term 5 (APS4322-7000)/APS Outputs/Current Q 3X0 <-> Data Pointer/QCurrentSetPoints[18]
//     Term 5 (APS4322-7000)/APS Outputs/Current Q 3X1 <-> Data Pointer/QCurrentSetPoints[19]
//     Term 5 (APS4322-7000)/APS Outputs/Current Q 3X2 <-> Data Pointer/QCurrentSetPoints[20]
//     Term 5 (APS4322-7000)/APS Outputs/Current Q 0Y0 <-> Data Pointer/QCurrentSetPoints[3]
//     Term 5 (APS4322-7000)/APS Outputs/Current Q 0Y1 <-> Data Pointer/QCurrentSetPoints[4]
//     Term 5 (APS4322-7000)/APS Outputs/Current Q 0Y2 <-> Data Pointer/QCurrentSetPoints[5]
//     Term 5 (APS4322-7000)/APS Outputs/Current Q 1Y0 <-> Data Pointer/QCurrentSetPoints[9]
//     Term 5 (APS4322-7000)/APS Outputs/Current Q 1Y1 <-> Data Pointer/QCurrentSetPoints[10]
//     Term 5 (APS4322-7000)/APS Outputs/Current Q 1Y2 <-> Data Pointer/QCurrentSetPoints[11]
//     Term 5 (APS4322-7000)/APS Outputs/Current Q 2Y0 <-> Data Pointer/QCurrentSetPoints[15]
//     Term 5 (APS4322-7000)/APS Outputs/Current Q 2Y1 <-> Data Pointer/QCurrentSetPoints[16]
//     Term 5 (APS4322-7000)/APS Outputs/Current Q 2Y2 <-> Data Pointer/QCurrentSetPoints[17]
//     Term 5 (APS4322-7000)/APS Outputs/Current Q 3Y0 <-> Data Pointer/QCurrentSetPoints[21]
//     Term 5 (APS4322-7000)/APS Outputs/Current Q 3Y1 <-> Data Pointer/QCurrentSetPoints[22]
//     Term 5 (APS4322-7000)/APS Outputs/Current Q 3Y2 <-> Data Pointer/QCurrentSetPoints[23]
//     Term 5 (APS4322-7000)/APS Outputs/PhiE 0X0 <-> Data Pointer/PhiSetPoints[0]
//     Term 5 (APS4322-7000)/APS Outputs/PhiE 0X1 <-> Data Pointer/PhiSetPoints[1]
//     Term 5 (APS4322-7000)/APS Outputs/PhiE 0X2 <-> Data Pointer/PhiSetPoints[2]
//     Term 5 (APS4322-7000)/APS Outputs/PhiE 1X0 <-> Data Pointer/PhiSetPoints[6]
//     Term 5 (APS4322-7000)/APS Outputs/PhiE 1X1 <-> Data Pointer/PhiSetPoints[7]
//     Term 5 (APS4322-7000)/APS Outputs/PhiE 1X2 <-> Data Pointer/PhiSetPoints[8]
//     Term 5 (APS4322-7000)/APS Outputs/PhiE 2X0 <-> Data Pointer/PhiSetPoints[12]
//     Term 5 (APS4322-7000)/APS Outputs/PhiE 2X1 <-> Data Pointer/PhiSetPoints[13]
//     Term 5 (APS4322-7000)/APS Outputs/PhiE 2X2 <-> Data Pointer/PhiSetPoints[14]
//     Term 5 (APS4322-7000)/APS Outputs/PhiE 3X0 <-> Data Pointer/PhiSetPoints[18]
//     Term 5 (APS4322-7000)/APS Outputs/PhiE 3X1 <-> Data Pointer/PhiSetPoints[19]
//     Term 5 (APS4322-7000)/APS Outputs/PhiE 3X2 <-> Data Pointer/PhiSetPoints[20]
//     Term 5 (APS4322-7000)/APS Outputs/PhiE 0Y0 <-> Data Pointer/PhiSetPoints[3]
//     Term 5 (APS4322-7000)/APS Outputs/PhiE 0Y1 <-> Data Pointer/PhiSetPoints[4]
//     Term 5 (APS4322-7000)/APS Outputs/PhiE 0Y2 <-> Data Pointer/PhiSetPoints[5]
//     Term 5 (APS4322-7000)/APS Outputs/PhiE 1Y0 <-> Data Pointer/PhiSetPoints[9]
//     Term 5 (APS4322-7000)/APS Outputs/PhiE 1Y1 <-> Data Pointer/PhiSetPoints[10]
//     Term 5 (APS4322-7000)/APS Outputs/PhiE 1Y2 <-> Data Pointer/PhiSetPoints[11]
//     Term 5 (APS4322-7000)/APS Outputs/PhiE 2Y0 <-> Data Pointer/PhiSetPoints[15]
//     Term 5 (APS4322-7000)/APS Outputs/PhiE 2Y1 <-> Data Pointer/PhiSetPoints[16]
//     Term 5 (APS4322-7000)/APS Outputs/PhiE 2Y2 <-> Data Pointer/PhiSetPoints[17]
//     Term 5 (APS4322-7000)/APS Outputs/PhiE 3Y0 <-> Data Pointer/PhiSetPoints[21]
//     Term 5 (APS4322-7000)/APS Outputs/PhiE 3Y1 <-> Data Pointer/PhiSetPoints[22]
//     Term 5 (APS4322-7000)/APS Outputs/PhiE 3Y2 <-> Data Pointer/PhiSetPoints[23]
//     Term 5 (APS4322-7000)/Term 6 (APS4322-5000)/FB Inputs/A{0..8 step 2} X-Field <-> Data Pointer/HallSensorFieldsXYZ[{0..12 step 3}]  (5 links)
//     Term 5 (APS4322-7000)/Term 6 (APS4322-5000)/FB Inputs/A{0..8 step 2} Y-Field <-> Data Pointer/HallSensorFieldsXYZ[{1..13 step 3}]  (5 links)
//     Term 5 (APS4322-7000)/Term 6 (APS4322-5000)/FB Inputs/A{0..8 step 2} Z-Field <-> Data Pointer/HallSensorFieldsXYZ[{2..14 step 3}]  (5 links)
//     Term 5 (APS4322-7000)/Term 6 (APS4322-5000)/FB Inputs/B{1..9 step 2} X-Field <-> Data Pointer/HallSensorFieldsXYZ[{15..27 step 3}]  (5 links)
//     Term 5 (APS4322-7000)/Term 6 (APS4322-5000)/FB Inputs/B{1..9 step 2} Y-Field <-> Data Pointer/HallSensorFieldsXYZ[{16..28 step 3}]  (5 links)
//     Term 5 (APS4322-7000)/Term 6 (APS4322-5000)/FB Inputs/B{1..9 step 2} Z-Field <-> Data Pointer/HallSensorFieldsXYZ[{17..29 step 3}]  (5 links)
//     Term 5 (APS4322-7000)/Term 6 (APS4322-5000)/FB Inputs/C{0..8 step 2} X-Field <-> Data Pointer/HallSensorFieldsXYZ[{30..42 step 3}]  (5 links)
//     Term 5 (APS4322-7000)/Term 6 (APS4322-5000)/FB Inputs/C{0..8 step 2} Y-Field <-> Data Pointer/HallSensorFieldsXYZ[{31..43 step 3}]  (5 links)
//     Term 5 (APS4322-7000)/Term 6 (APS4322-5000)/FB Inputs/C{0..8 step 2} Z-Field <-> Data Pointer/HallSensorFieldsXYZ[{32..44 step 3}]  (5 links)
//     Term 5 (APS4322-7000)/Term 6 (APS4322-5000)/FB Inputs/D{1..9 step 2} X-Field <-> Data Pointer/HallSensorFieldsXYZ[{45..57 step 3}]  (5 links)
//     Term 5 (APS4322-7000)/Term 6 (APS4322-5000)/FB Inputs/D{1..9 step 2} Y-Field <-> Data Pointer/HallSensorFieldsXYZ[{46..58 step 3}]  (5 links)
//     Term 5 (APS4322-7000)/Term 6 (APS4322-5000)/FB Inputs/D{1..9 step 2} Z-Field <-> Data Pointer/HallSensorFieldsXYZ[{47..59 step 3}]  (5 links)
//     Term 5 (APS4322-7000)/Term 6 (APS4322-5000)/FB Inputs/E{0..8 step 2} X-Field <-> Data Pointer/HallSensorFieldsXYZ[{60..72 step 3}]  (5 links)
//     Term 5 (APS4322-7000)/Term 6 (APS4322-5000)/FB Inputs/E{0..8 step 2} Y-Field <-> Data Pointer/HallSensorFieldsXYZ[{61..73 step 3}]  (5 links)
//     Term 5 (APS4322-7000)/Term 6 (APS4322-5000)/FB Inputs/E{0..8 step 2} Z-Field <-> Data Pointer/HallSensorFieldsXYZ[{62..74 step 3}]  (5 links)
//     Term 5 (APS4322-7000)/Term 6 (APS4322-5000)/FB Inputs/F{1..9 step 2} X-Field <-> Data Pointer/HallSensorFieldsXYZ[{75..87 step 3}]  (5 links)
//     Term 5 (APS4322-7000)/Term 6 (APS4322-5000)/FB Inputs/F{1..9 step 2} Y-Field <-> Data Pointer/HallSensorFieldsXYZ[{76..88 step 3}]  (5 links)
//     Term 5 (APS4322-7000)/Term 6 (APS4322-5000)/FB Inputs/F{1..9 step 2} Z-Field <-> Data Pointer/HallSensorFieldsXYZ[{77..89 step 3}]  (5 links)
//     Term 5 (APS4322-7000)/Term 6 (APS4322-5000)/FB Inputs/G{0..8 step 2} X-Field <-> Data Pointer/HallSensorFieldsXYZ[{90..102 step 3}]  (5 links)
//     Term 5 (APS4322-7000)/Term 6 (APS4322-5000)/FB Inputs/G{0..8 step 2} Y-Field <-> Data Pointer/HallSensorFieldsXYZ[{91..103 step 3}]  (5 links)
//     Term 5 (APS4322-7000)/Term 6 (APS4322-5000)/FB Inputs/G{0..8 step 2} Z-Field <-> Data Pointer/HallSensorFieldsXYZ[{92..104 step 3}]  (5 links)
//     Term 5 (APS4322-7000)/Term 6 (APS4322-5000)/FB Inputs/H{1..9 step 2} X-Field <-> Data Pointer/HallSensorFieldsXYZ[{105..117 step 3}]  (5 links)
//     Term 5 (APS4322-7000)/Term 6 (APS4322-5000)/FB Inputs/H{1..9 step 2} Y-Field <-> Data Pointer/HallSensorFieldsXYZ[{106..118 step 3}]  (5 links)
//     Term 5 (APS4322-7000)/Term 6 (APS4322-5000)/FB Inputs/H{1..9 step 2} Z-Field <-> Data Pointer/HallSensorFieldsXYZ[{107..119 step 3}]  (5 links)
//     Term 5 (APS4322-7000)/Term 6 (APS4322-5000)/FB Inputs/I{0..8 step 2} X-Field <-> Data Pointer/HallSensorFieldsXYZ[{120..132 step 3}]  (5 links)
//     Term 5 (APS4322-7000)/Term 6 (APS4322-5000)/FB Inputs/I{0..8 step 2} Y-Field <-> Data Pointer/HallSensorFieldsXYZ[{121..133 step 3}]  (5 links)
//     Term 5 (APS4322-7000)/Term 6 (APS4322-5000)/FB Inputs/I{0..8 step 2} Z-Field <-> Data Pointer/HallSensorFieldsXYZ[{122..134 step 3}]  (5 links)
//     Term 5 (APS4322-7000)/Term 6 (APS4322-5000)/FB Inputs/J{1..9 step 2} X-Field <-> Data Pointer/HallSensorFieldsXYZ[{135..147 step 3}]  (5 links)
//     Term 5 (APS4322-7000)/Term 6 (APS4322-5000)/FB Inputs/J{1..9 step 2} Y-Field <-> Data Pointer/HallSensorFieldsXYZ[{136..148 step 3}]  (5 links)
//     Term 5 (APS4322-7000)/Term 6 (APS4322-5000)/FB Inputs/J{1..9 step 2} Z-Field <-> Data Pointer/HallSensorFieldsXYZ[{137..149 step 3}]  (5 links)
//     Term 5 (APS4322-7000)/Term 6 (APS4322-5000)/FB Inputs/Status <-> Data Pointer/FeedbackStatus
//   Device 2 (EtherCAT) <-> TcCOM Objects/XPlanar/Part1/APS4322_P1_4
//     Term 7 (APS4322-7000)/APS Comm Inputs/CommStatusWord <-> Data Pointer/MoverCommStatusWord
//     Term 7 (APS4322-7000)/APS Comm Inputs/Data {1..4} <-> Data Pointer/MoverCommDataIn[{0..3}]  (4 links)
//     Term 7 (APS4322-7000)/APS Comm Outputs/CommControlWord <-> Data Pointer/MoverCommControlWord
//     Term 7 (APS4322-7000)/APS Comm Outputs/Data 1 <-> Data Pointer/MoverCommDataOut
//     Term 7 (APS4322-7000)/APS Diagdata/DC Link Voltage <-> Data Pointer/DcLinkVoltage
//     Term 7 (APS4322-7000)/APS Diagdata/Power supply current <-> Data Pointer/PowerSupplyCurrent
//     Term 7 (APS4322-7000)/APS Inputs/StatusWord <-> Data Pointer/PowerUnitStatusWord
//     Term 7 (APS4322-7000)/APS Outputs/ControlWord <-> Data Pointer/PowerUnitControlWord
//     Term 7 (APS4322-7000)/APS Outputs/Current D 0X0 <-> Data Pointer/DCurrentSetPoints[0]
//     Term 7 (APS4322-7000)/APS Outputs/Current D 0X1 <-> Data Pointer/DCurrentSetPoints[1]
//     Term 7 (APS4322-7000)/APS Outputs/Current D 0X2 <-> Data Pointer/DCurrentSetPoints[2]
//     Term 7 (APS4322-7000)/APS Outputs/Current D 1X0 <-> Data Pointer/DCurrentSetPoints[6]
//     Term 7 (APS4322-7000)/APS Outputs/Current D 1X1 <-> Data Pointer/DCurrentSetPoints[7]
//     Term 7 (APS4322-7000)/APS Outputs/Current D 1X2 <-> Data Pointer/DCurrentSetPoints[8]
//     Term 7 (APS4322-7000)/APS Outputs/Current D 2X0 <-> Data Pointer/DCurrentSetPoints[12]
//     Term 7 (APS4322-7000)/APS Outputs/Current D 2X1 <-> Data Pointer/DCurrentSetPoints[13]
//     Term 7 (APS4322-7000)/APS Outputs/Current D 2X2 <-> Data Pointer/DCurrentSetPoints[14]
//     Term 7 (APS4322-7000)/APS Outputs/Current D 3X0 <-> Data Pointer/DCurrentSetPoints[18]
//     Term 7 (APS4322-7000)/APS Outputs/Current D 3X1 <-> Data Pointer/DCurrentSetPoints[19]
//     Term 7 (APS4322-7000)/APS Outputs/Current D 3X2 <-> Data Pointer/DCurrentSetPoints[20]
//     Term 7 (APS4322-7000)/APS Outputs/Current D 0Y0 <-> Data Pointer/DCurrentSetPoints[3]
//     Term 7 (APS4322-7000)/APS Outputs/Current D 0Y1 <-> Data Pointer/DCurrentSetPoints[4]
//     Term 7 (APS4322-7000)/APS Outputs/Current D 0Y2 <-> Data Pointer/DCurrentSetPoints[5]
//     Term 7 (APS4322-7000)/APS Outputs/Current D 1Y0 <-> Data Pointer/DCurrentSetPoints[9]
//     Term 7 (APS4322-7000)/APS Outputs/Current D 1Y1 <-> Data Pointer/DCurrentSetPoints[10]
//     Term 7 (APS4322-7000)/APS Outputs/Current D 1Y2 <-> Data Pointer/DCurrentSetPoints[11]
//     Term 7 (APS4322-7000)/APS Outputs/Current D 2Y0 <-> Data Pointer/DCurrentSetPoints[15]
//     Term 7 (APS4322-7000)/APS Outputs/Current D 2Y1 <-> Data Pointer/DCurrentSetPoints[16]
//     Term 7 (APS4322-7000)/APS Outputs/Current D 2Y2 <-> Data Pointer/DCurrentSetPoints[17]
//     Term 7 (APS4322-7000)/APS Outputs/Current D 3Y0 <-> Data Pointer/DCurrentSetPoints[21]
//     Term 7 (APS4322-7000)/APS Outputs/Current D 3Y1 <-> Data Pointer/DCurrentSetPoints[22]
//     Term 7 (APS4322-7000)/APS Outputs/Current D 3Y2 <-> Data Pointer/DCurrentSetPoints[23]
//     Term 7 (APS4322-7000)/APS Outputs/Current Q 0X0 <-> Data Pointer/QCurrentSetPoints[0]
//     Term 7 (APS4322-7000)/APS Outputs/Current Q 0X1 <-> Data Pointer/QCurrentSetPoints[1]
//     Term 7 (APS4322-7000)/APS Outputs/Current Q 0X2 <-> Data Pointer/QCurrentSetPoints[2]
//     Term 7 (APS4322-7000)/APS Outputs/Current Q 1X0 <-> Data Pointer/QCurrentSetPoints[6]
//     Term 7 (APS4322-7000)/APS Outputs/Current Q 1X1 <-> Data Pointer/QCurrentSetPoints[7]
//     Term 7 (APS4322-7000)/APS Outputs/Current Q 1X2 <-> Data Pointer/QCurrentSetPoints[8]
//     Term 7 (APS4322-7000)/APS Outputs/Current Q 2X0 <-> Data Pointer/QCurrentSetPoints[12]
//     Term 7 (APS4322-7000)/APS Outputs/Current Q 2X1 <-> Data Pointer/QCurrentSetPoints[13]
//     Term 7 (APS4322-7000)/APS Outputs/Current Q 2X2 <-> Data Pointer/QCurrentSetPoints[14]
//     Term 7 (APS4322-7000)/APS Outputs/Current Q 3X0 <-> Data Pointer/QCurrentSetPoints[18]
//     Term 7 (APS4322-7000)/APS Outputs/Current Q 3X1 <-> Data Pointer/QCurrentSetPoints[19]
//     Term 7 (APS4322-7000)/APS Outputs/Current Q 3X2 <-> Data Pointer/QCurrentSetPoints[20]
//     Term 7 (APS4322-7000)/APS Outputs/Current Q 0Y0 <-> Data Pointer/QCurrentSetPoints[3]
//     Term 7 (APS4322-7000)/APS Outputs/Current Q 0Y1 <-> Data Pointer/QCurrentSetPoints[4]
//     Term 7 (APS4322-7000)/APS Outputs/Current Q 0Y2 <-> Data Pointer/QCurrentSetPoints[5]
//     Term 7 (APS4322-7000)/APS Outputs/Current Q 1Y0 <-> Data Pointer/QCurrentSetPoints[9]
//     Term 7 (APS4322-7000)/APS Outputs/Current Q 1Y1 <-> Data Pointer/QCurrentSetPoints[10]
//     Term 7 (APS4322-7000)/APS Outputs/Current Q 1Y2 <-> Data Pointer/QCurrentSetPoints[11]
//     Term 7 (APS4322-7000)/APS Outputs/Current Q 2Y0 <-> Data Pointer/QCurrentSetPoints[15]
//     Term 7 (APS4322-7000)/APS Outputs/Current Q 2Y1 <-> Data Pointer/QCurrentSetPoints[16]
//     Term 7 (APS4322-7000)/APS Outputs/Current Q 2Y2 <-> Data Pointer/QCurrentSetPoints[17]
//     Term 7 (APS4322-7000)/APS Outputs/Current Q 3Y0 <-> Data Pointer/QCurrentSetPoints[21]
//     Term 7 (APS4322-7000)/APS Outputs/Current Q 3Y1 <-> Data Pointer/QCurrentSetPoints[22]
//     Term 7 (APS4322-7000)/APS Outputs/Current Q 3Y2 <-> Data Pointer/QCurrentSetPoints[23]
//     Term 7 (APS4322-7000)/APS Outputs/PhiE 0X0 <-> Data Pointer/PhiSetPoints[0]
//     Term 7 (APS4322-7000)/APS Outputs/PhiE 0X1 <-> Data Pointer/PhiSetPoints[1]
//     Term 7 (APS4322-7000)/APS Outputs/PhiE 0X2 <-> Data Pointer/PhiSetPoints[2]
//     Term 7 (APS4322-7000)/APS Outputs/PhiE 1X0 <-> Data Pointer/PhiSetPoints[6]
//     Term 7 (APS4322-7000)/APS Outputs/PhiE 1X1 <-> Data Pointer/PhiSetPoints[7]
//     Term 7 (APS4322-7000)/APS Outputs/PhiE 1X2 <-> Data Pointer/PhiSetPoints[8]
//     Term 7 (APS4322-7000)/APS Outputs/PhiE 2X0 <-> Data Pointer/PhiSetPoints[12]
//     Term 7 (APS4322-7000)/APS Outputs/PhiE 2X1 <-> Data Pointer/PhiSetPoints[13]
//     Term 7 (APS4322-7000)/APS Outputs/PhiE 2X2 <-> Data Pointer/PhiSetPoints[14]
//     Term 7 (APS4322-7000)/APS Outputs/PhiE 3X0 <-> Data Pointer/PhiSetPoints[18]
//     Term 7 (APS4322-7000)/APS Outputs/PhiE 3X1 <-> Data Pointer/PhiSetPoints[19]
//     Term 7 (APS4322-7000)/APS Outputs/PhiE 3X2 <-> Data Pointer/PhiSetPoints[20]
//     Term 7 (APS4322-7000)/APS Outputs/PhiE 0Y0 <-> Data Pointer/PhiSetPoints[3]
//     Term 7 (APS4322-7000)/APS Outputs/PhiE 0Y1 <-> Data Pointer/PhiSetPoints[4]
//     Term 7 (APS4322-7000)/APS Outputs/PhiE 0Y2 <-> Data Pointer/PhiSetPoints[5]
//     Term 7 (APS4322-7000)/APS Outputs/PhiE 1Y0 <-> Data Pointer/PhiSetPoints[9]
//     Term 7 (APS4322-7000)/APS Outputs/PhiE 1Y1 <-> Data Pointer/PhiSetPoints[10]
//     Term 7 (APS4322-7000)/APS Outputs/PhiE 1Y2 <-> Data Pointer/PhiSetPoints[11]
//     Term 7 (APS4322-7000)/APS Outputs/PhiE 2Y0 <-> Data Pointer/PhiSetPoints[15]
//     Term 7 (APS4322-7000)/APS Outputs/PhiE 2Y1 <-> Data Pointer/PhiSetPoints[16]
//     Term 7 (APS4322-7000)/APS Outputs/PhiE 2Y2 <-> Data Pointer/PhiSetPoints[17]
//     Term 7 (APS4322-7000)/APS Outputs/PhiE 3Y0 <-> Data Pointer/PhiSetPoints[21]
//     Term 7 (APS4322-7000)/APS Outputs/PhiE 3Y1 <-> Data Pointer/PhiSetPoints[22]
//     Term 7 (APS4322-7000)/APS Outputs/PhiE 3Y2 <-> Data Pointer/PhiSetPoints[23]
//     Term 7 (APS4322-7000)/Term 8 (APS4322-5000)/FB Inputs/A{0..8 step 2} X-Field <-> Data Pointer/HallSensorFieldsXYZ[{0..12 step 3}]  (5 links)
//     Term 7 (APS4322-7000)/Term 8 (APS4322-5000)/FB Inputs/A{0..8 step 2} Y-Field <-> Data Pointer/HallSensorFieldsXYZ[{1..13 step 3}]  (5 links)
//     Term 7 (APS4322-7000)/Term 8 (APS4322-5000)/FB Inputs/A{0..8 step 2} Z-Field <-> Data Pointer/HallSensorFieldsXYZ[{2..14 step 3}]  (5 links)
//     Term 7 (APS4322-7000)/Term 8 (APS4322-5000)/FB Inputs/B{1..9 step 2} X-Field <-> Data Pointer/HallSensorFieldsXYZ[{15..27 step 3}]  (5 links)
//     Term 7 (APS4322-7000)/Term 8 (APS4322-5000)/FB Inputs/B{1..9 step 2} Y-Field <-> Data Pointer/HallSensorFieldsXYZ[{16..28 step 3}]  (5 links)
//     Term 7 (APS4322-7000)/Term 8 (APS4322-5000)/FB Inputs/B{1..9 step 2} Z-Field <-> Data Pointer/HallSensorFieldsXYZ[{17..29 step 3}]  (5 links)
//     Term 7 (APS4322-7000)/Term 8 (APS4322-5000)/FB Inputs/C{0..8 step 2} X-Field <-> Data Pointer/HallSensorFieldsXYZ[{30..42 step 3}]  (5 links)
//     Term 7 (APS4322-7000)/Term 8 (APS4322-5000)/FB Inputs/C{0..8 step 2} Y-Field <-> Data Pointer/HallSensorFieldsXYZ[{31..43 step 3}]  (5 links)
//     Term 7 (APS4322-7000)/Term 8 (APS4322-5000)/FB Inputs/C{0..8 step 2} Z-Field <-> Data Pointer/HallSensorFieldsXYZ[{32..44 step 3}]  (5 links)
//     Term 7 (APS4322-7000)/Term 8 (APS4322-5000)/FB Inputs/D{1..9 step 2} X-Field <-> Data Pointer/HallSensorFieldsXYZ[{45..57 step 3}]  (5 links)
//     Term 7 (APS4322-7000)/Term 8 (APS4322-5000)/FB Inputs/D{1..9 step 2} Y-Field <-> Data Pointer/HallSensorFieldsXYZ[{46..58 step 3}]  (5 links)
//     Term 7 (APS4322-7000)/Term 8 (APS4322-5000)/FB Inputs/D{1..9 step 2} Z-Field <-> Data Pointer/HallSensorFieldsXYZ[{47..59 step 3}]  (5 links)
//     Term 7 (APS4322-7000)/Term 8 (APS4322-5000)/FB Inputs/E{0..8 step 2} X-Field <-> Data Pointer/HallSensorFieldsXYZ[{60..72 step 3}]  (5 links)
//     Term 7 (APS4322-7000)/Term 8 (APS4322-5000)/FB Inputs/E{0..8 step 2} Y-Field <-> Data Pointer/HallSensorFieldsXYZ[{61..73 step 3}]  (5 links)
//     Term 7 (APS4322-7000)/Term 8 (APS4322-5000)/FB Inputs/E{0..8 step 2} Z-Field <-> Data Pointer/HallSensorFieldsXYZ[{62..74 step 3}]  (5 links)
//     Term 7 (APS4322-7000)/Term 8 (APS4322-5000)/FB Inputs/F{1..9 step 2} X-Field <-> Data Pointer/HallSensorFieldsXYZ[{75..87 step 3}]  (5 links)
//     Term 7 (APS4322-7000)/Term 8 (APS4322-5000)/FB Inputs/F{1..9 step 2} Y-Field <-> Data Pointer/HallSensorFieldsXYZ[{76..88 step 3}]  (5 links)
//     Term 7 (APS4322-7000)/Term 8 (APS4322-5000)/FB Inputs/F{1..9 step 2} Z-Field <-> Data Pointer/HallSensorFieldsXYZ[{77..89 step 3}]  (5 links)
//     Term 7 (APS4322-7000)/Term 8 (APS4322-5000)/FB Inputs/G{0..8 step 2} X-Field <-> Data Pointer/HallSensorFieldsXYZ[{90..102 step 3}]  (5 links)
//     Term 7 (APS4322-7000)/Term 8 (APS4322-5000)/FB Inputs/G{0..8 step 2} Y-Field <-> Data Pointer/HallSensorFieldsXYZ[{91..103 step 3}]  (5 links)
//     Term 7 (APS4322-7000)/Term 8 (APS4322-5000)/FB Inputs/G{0..8 step 2} Z-Field <-> Data Pointer/HallSensorFieldsXYZ[{92..104 step 3}]  (5 links)
//     Term 7 (APS4322-7000)/Term 8 (APS4322-5000)/FB Inputs/H{1..9 step 2} X-Field <-> Data Pointer/HallSensorFieldsXYZ[{105..117 step 3}]  (5 links)
//     Term 7 (APS4322-7000)/Term 8 (APS4322-5000)/FB Inputs/H{1..9 step 2} Y-Field <-> Data Pointer/HallSensorFieldsXYZ[{106..118 step 3}]  (5 links)
//     Term 7 (APS4322-7000)/Term 8 (APS4322-5000)/FB Inputs/H{1..9 step 2} Z-Field <-> Data Pointer/HallSensorFieldsXYZ[{107..119 step 3}]  (5 links)
//     Term 7 (APS4322-7000)/Term 8 (APS4322-5000)/FB Inputs/I{0..8 step 2} X-Field <-> Data Pointer/HallSensorFieldsXYZ[{120..132 step 3}]  (5 links)
//     Term 7 (APS4322-7000)/Term 8 (APS4322-5000)/FB Inputs/I{0..8 step 2} Y-Field <-> Data Pointer/HallSensorFieldsXYZ[{121..133 step 3}]  (5 links)
//     Term 7 (APS4322-7000)/Term 8 (APS4322-5000)/FB Inputs/I{0..8 step 2} Z-Field <-> Data Pointer/HallSensorFieldsXYZ[{122..134 step 3}]  (5 links)
//     Term 7 (APS4322-7000)/Term 8 (APS4322-5000)/FB Inputs/J{1..9 step 2} X-Field <-> Data Pointer/HallSensorFieldsXYZ[{135..147 step 3}]  (5 links)
//     Term 7 (APS4322-7000)/Term 8 (APS4322-5000)/FB Inputs/J{1..9 step 2} Y-Field <-> Data Pointer/HallSensorFieldsXYZ[{136..148 step 3}]  (5 links)
//     Term 7 (APS4322-7000)/Term 8 (APS4322-5000)/FB Inputs/J{1..9 step 2} Z-Field <-> Data Pointer/HallSensorFieldsXYZ[{137..149 step 3}]  (5 links)
//     Term 7 (APS4322-7000)/Term 8 (APS4322-5000)/FB Inputs/Status <-> Data Pointer/FeedbackStatus
//   Device 2 (EtherCAT) <-> TcCOM Objects/XPlanar/Part1/APS4322_P1_5
//     Term 9 (APS4322-7000)/APS Comm Inputs/CommStatusWord <-> Data Pointer/MoverCommStatusWord
//     Term 9 (APS4322-7000)/APS Comm Inputs/Data {1..4} <-> Data Pointer/MoverCommDataIn[{0..3}]  (4 links)
//     Term 9 (APS4322-7000)/APS Comm Outputs/CommControlWord <-> Data Pointer/MoverCommControlWord
//     Term 9 (APS4322-7000)/APS Comm Outputs/Data 1 <-> Data Pointer/MoverCommDataOut
//     Term 9 (APS4322-7000)/APS Diagdata/DC Link Voltage <-> Data Pointer/DcLinkVoltage
//     Term 9 (APS4322-7000)/APS Diagdata/Power supply current <-> Data Pointer/PowerSupplyCurrent
//     Term 9 (APS4322-7000)/APS Inputs/StatusWord <-> Data Pointer/PowerUnitStatusWord
//     Term 9 (APS4322-7000)/APS Outputs/ControlWord <-> Data Pointer/PowerUnitControlWord
//     Term 9 (APS4322-7000)/APS Outputs/Current D 0X0 <-> Data Pointer/DCurrentSetPoints[0]
//     Term 9 (APS4322-7000)/APS Outputs/Current D 0X1 <-> Data Pointer/DCurrentSetPoints[1]
//     Term 9 (APS4322-7000)/APS Outputs/Current D 0X2 <-> Data Pointer/DCurrentSetPoints[2]
//     Term 9 (APS4322-7000)/APS Outputs/Current D 1X0 <-> Data Pointer/DCurrentSetPoints[6]
//     Term 9 (APS4322-7000)/APS Outputs/Current D 1X1 <-> Data Pointer/DCurrentSetPoints[7]
//     Term 9 (APS4322-7000)/APS Outputs/Current D 1X2 <-> Data Pointer/DCurrentSetPoints[8]
//     Term 9 (APS4322-7000)/APS Outputs/Current D 2X0 <-> Data Pointer/DCurrentSetPoints[12]
//     Term 9 (APS4322-7000)/APS Outputs/Current D 2X1 <-> Data Pointer/DCurrentSetPoints[13]
//     Term 9 (APS4322-7000)/APS Outputs/Current D 2X2 <-> Data Pointer/DCurrentSetPoints[14]
//     Term 9 (APS4322-7000)/APS Outputs/Current D 3X0 <-> Data Pointer/DCurrentSetPoints[18]
//     Term 9 (APS4322-7000)/APS Outputs/Current D 3X1 <-> Data Pointer/DCurrentSetPoints[19]
//     Term 9 (APS4322-7000)/APS Outputs/Current D 3X2 <-> Data Pointer/DCurrentSetPoints[20]
//     Term 9 (APS4322-7000)/APS Outputs/Current D 0Y0 <-> Data Pointer/DCurrentSetPoints[3]
//     Term 9 (APS4322-7000)/APS Outputs/Current D 0Y1 <-> Data Pointer/DCurrentSetPoints[4]
//     Term 9 (APS4322-7000)/APS Outputs/Current D 0Y2 <-> Data Pointer/DCurrentSetPoints[5]
//     Term 9 (APS4322-7000)/APS Outputs/Current D 1Y0 <-> Data Pointer/DCurrentSetPoints[9]
//     Term 9 (APS4322-7000)/APS Outputs/Current D 1Y1 <-> Data Pointer/DCurrentSetPoints[10]
//     Term 9 (APS4322-7000)/APS Outputs/Current D 1Y2 <-> Data Pointer/DCurrentSetPoints[11]
//     Term 9 (APS4322-7000)/APS Outputs/Current D 2Y0 <-> Data Pointer/DCurrentSetPoints[15]
//     Term 9 (APS4322-7000)/APS Outputs/Current D 2Y1 <-> Data Pointer/DCurrentSetPoints[16]
//     Term 9 (APS4322-7000)/APS Outputs/Current D 2Y2 <-> Data Pointer/DCurrentSetPoints[17]
//     Term 9 (APS4322-7000)/APS Outputs/Current D 3Y0 <-> Data Pointer/DCurrentSetPoints[21]
//     Term 9 (APS4322-7000)/APS Outputs/Current D 3Y1 <-> Data Pointer/DCurrentSetPoints[22]
//     Term 9 (APS4322-7000)/APS Outputs/Current D 3Y2 <-> Data Pointer/DCurrentSetPoints[23]
//     Term 9 (APS4322-7000)/APS Outputs/Current Q 0X0 <-> Data Pointer/QCurrentSetPoints[0]
//     Term 9 (APS4322-7000)/APS Outputs/Current Q 0X1 <-> Data Pointer/QCurrentSetPoints[1]
//     Term 9 (APS4322-7000)/APS Outputs/Current Q 0X2 <-> Data Pointer/QCurrentSetPoints[2]
//     Term 9 (APS4322-7000)/APS Outputs/Current Q 1X0 <-> Data Pointer/QCurrentSetPoints[6]
//     Term 9 (APS4322-7000)/APS Outputs/Current Q 1X1 <-> Data Pointer/QCurrentSetPoints[7]
//     Term 9 (APS4322-7000)/APS Outputs/Current Q 1X2 <-> Data Pointer/QCurrentSetPoints[8]
//     Term 9 (APS4322-7000)/APS Outputs/Current Q 2X0 <-> Data Pointer/QCurrentSetPoints[12]
//     Term 9 (APS4322-7000)/APS Outputs/Current Q 2X1 <-> Data Pointer/QCurrentSetPoints[13]
//     Term 9 (APS4322-7000)/APS Outputs/Current Q 2X2 <-> Data Pointer/QCurrentSetPoints[14]
//     Term 9 (APS4322-7000)/APS Outputs/Current Q 3X0 <-> Data Pointer/QCurrentSetPoints[18]
//     Term 9 (APS4322-7000)/APS Outputs/Current Q 3X1 <-> Data Pointer/QCurrentSetPoints[19]
//     Term 9 (APS4322-7000)/APS Outputs/Current Q 3X2 <-> Data Pointer/QCurrentSetPoints[20]
//     Term 9 (APS4322-7000)/APS Outputs/Current Q 0Y0 <-> Data Pointer/QCurrentSetPoints[3]
//     Term 9 (APS4322-7000)/APS Outputs/Current Q 0Y1 <-> Data Pointer/QCurrentSetPoints[4]
//     Term 9 (APS4322-7000)/APS Outputs/Current Q 0Y2 <-> Data Pointer/QCurrentSetPoints[5]
//     Term 9 (APS4322-7000)/APS Outputs/Current Q 1Y0 <-> Data Pointer/QCurrentSetPoints[9]
//     Term 9 (APS4322-7000)/APS Outputs/Current Q 1Y1 <-> Data Pointer/QCurrentSetPoints[10]
//     Term 9 (APS4322-7000)/APS Outputs/Current Q 1Y2 <-> Data Pointer/QCurrentSetPoints[11]
//     Term 9 (APS4322-7000)/APS Outputs/Current Q 2Y0 <-> Data Pointer/QCurrentSetPoints[15]
//     Term 9 (APS4322-7000)/APS Outputs/Current Q 2Y1 <-> Data Pointer/QCurrentSetPoints[16]
//     Term 9 (APS4322-7000)/APS Outputs/Current Q 2Y2 <-> Data Pointer/QCurrentSetPoints[17]
//     Term 9 (APS4322-7000)/APS Outputs/Current Q 3Y0 <-> Data Pointer/QCurrentSetPoints[21]
//     Term 9 (APS4322-7000)/APS Outputs/Current Q 3Y1 <-> Data Pointer/QCurrentSetPoints[22]
//     Term 9 (APS4322-7000)/APS Outputs/Current Q 3Y2 <-> Data Pointer/QCurrentSetPoints[23]
//     Term 9 (APS4322-7000)/APS Outputs/PhiE 0X0 <-> Data Pointer/PhiSetPoints[0]
//     Term 9 (APS4322-7000)/APS Outputs/PhiE 0X1 <-> Data Pointer/PhiSetPoints[1]
//     Term 9 (APS4322-7000)/APS Outputs/PhiE 0X2 <-> Data Pointer/PhiSetPoints[2]
//     Term 9 (APS4322-7000)/APS Outputs/PhiE 1X0 <-> Data Pointer/PhiSetPoints[6]
//     Term 9 (APS4322-7000)/APS Outputs/PhiE 1X1 <-> Data Pointer/PhiSetPoints[7]
//     Term 9 (APS4322-7000)/APS Outputs/PhiE 1X2 <-> Data Pointer/PhiSetPoints[8]
//     Term 9 (APS4322-7000)/APS Outputs/PhiE 2X0 <-> Data Pointer/PhiSetPoints[12]
//     Term 9 (APS4322-7000)/APS Outputs/PhiE 2X1 <-> Data Pointer/PhiSetPoints[13]
//     Term 9 (APS4322-7000)/APS Outputs/PhiE 2X2 <-> Data Pointer/PhiSetPoints[14]
//     Term 9 (APS4322-7000)/APS Outputs/PhiE 3X0 <-> Data Pointer/PhiSetPoints[18]
//     Term 9 (APS4322-7000)/APS Outputs/PhiE 3X1 <-> Data Pointer/PhiSetPoints[19]
//     Term 9 (APS4322-7000)/APS Outputs/PhiE 3X2 <-> Data Pointer/PhiSetPoints[20]
//     Term 9 (APS4322-7000)/APS Outputs/PhiE 0Y0 <-> Data Pointer/PhiSetPoints[3]
//     Term 9 (APS4322-7000)/APS Outputs/PhiE 0Y1 <-> Data Pointer/PhiSetPoints[4]
//     Term 9 (APS4322-7000)/APS Outputs/PhiE 0Y2 <-> Data Pointer/PhiSetPoints[5]
//     Term 9 (APS4322-7000)/APS Outputs/PhiE 1Y0 <-> Data Pointer/PhiSetPoints[9]
//     Term 9 (APS4322-7000)/APS Outputs/PhiE 1Y1 <-> Data Pointer/PhiSetPoints[10]
//     Term 9 (APS4322-7000)/APS Outputs/PhiE 1Y2 <-> Data Pointer/PhiSetPoints[11]
//     Term 9 (APS4322-7000)/APS Outputs/PhiE 2Y0 <-> Data Pointer/PhiSetPoints[15]
//     Term 9 (APS4322-7000)/APS Outputs/PhiE 2Y1 <-> Data Pointer/PhiSetPoints[16]
//     Term 9 (APS4322-7000)/APS Outputs/PhiE 2Y2 <-> Data Pointer/PhiSetPoints[17]
//     Term 9 (APS4322-7000)/APS Outputs/PhiE 3Y0 <-> Data Pointer/PhiSetPoints[21]
//     Term 9 (APS4322-7000)/APS Outputs/PhiE 3Y1 <-> Data Pointer/PhiSetPoints[22]
//     Term 9 (APS4322-7000)/APS Outputs/PhiE 3Y2 <-> Data Pointer/PhiSetPoints[23]
//     Term 9 (APS4322-7000)/Term 10 (APS4322-5000)/FB Inputs/A{0..8 step 2} X-Field <-> Data Pointer/HallSensorFieldsXYZ[{0..12 step 3}]  (5 links)
//     Term 9 (APS4322-7000)/Term 10 (APS4322-5000)/FB Inputs/A{0..8 step 2} Y-Field <-> Data Pointer/HallSensorFieldsXYZ[{1..13 step 3}]  (5 links)
//     Term 9 (APS4322-7000)/Term 10 (APS4322-5000)/FB Inputs/A{0..8 step 2} Z-Field <-> Data Pointer/HallSensorFieldsXYZ[{2..14 step 3}]  (5 links)
//     Term 9 (APS4322-7000)/Term 10 (APS4322-5000)/FB Inputs/B{1..9 step 2} X-Field <-> Data Pointer/HallSensorFieldsXYZ[{15..27 step 3}]  (5 links)
//     Term 9 (APS4322-7000)/Term 10 (APS4322-5000)/FB Inputs/B{1..9 step 2} Y-Field <-> Data Pointer/HallSensorFieldsXYZ[{16..28 step 3}]  (5 links)
//     Term 9 (APS4322-7000)/Term 10 (APS4322-5000)/FB Inputs/B{1..9 step 2} Z-Field <-> Data Pointer/HallSensorFieldsXYZ[{17..29 step 3}]  (5 links)
//     Term 9 (APS4322-7000)/Term 10 (APS4322-5000)/FB Inputs/C{0..8 step 2} X-Field <-> Data Pointer/HallSensorFieldsXYZ[{30..42 step 3}]  (5 links)
//     Term 9 (APS4322-7000)/Term 10 (APS4322-5000)/FB Inputs/C{0..8 step 2} Y-Field <-> Data Pointer/HallSensorFieldsXYZ[{31..43 step 3}]  (5 links)
//     Term 9 (APS4322-7000)/Term 10 (APS4322-5000)/FB Inputs/C{0..8 step 2} Z-Field <-> Data Pointer/HallSensorFieldsXYZ[{32..44 step 3}]  (5 links)
//     Term 9 (APS4322-7000)/Term 10 (APS4322-5000)/FB Inputs/D{1..9 step 2} X-Field <-> Data Pointer/HallSensorFieldsXYZ[{45..57 step 3}]  (5 links)
//     Term 9 (APS4322-7000)/Term 10 (APS4322-5000)/FB Inputs/D{1..9 step 2} Y-Field <-> Data Pointer/HallSensorFieldsXYZ[{46..58 step 3}]  (5 links)
//     Term 9 (APS4322-7000)/Term 10 (APS4322-5000)/FB Inputs/D{1..9 step 2} Z-Field <-> Data Pointer/HallSensorFieldsXYZ[{47..59 step 3}]  (5 links)
//     Term 9 (APS4322-7000)/Term 10 (APS4322-5000)/FB Inputs/E{0..8 step 2} X-Field <-> Data Pointer/HallSensorFieldsXYZ[{60..72 step 3}]  (5 links)
//     Term 9 (APS4322-7000)/Term 10 (APS4322-5000)/FB Inputs/E{0..8 step 2} Y-Field <-> Data Pointer/HallSensorFieldsXYZ[{61..73 step 3}]  (5 links)
//     Term 9 (APS4322-7000)/Term 10 (APS4322-5000)/FB Inputs/E{0..8 step 2} Z-Field <-> Data Pointer/HallSensorFieldsXYZ[{62..74 step 3}]  (5 links)
//     Term 9 (APS4322-7000)/Term 10 (APS4322-5000)/FB Inputs/F{1..9 step 2} X-Field <-> Data Pointer/HallSensorFieldsXYZ[{75..87 step 3}]  (5 links)
//     Term 9 (APS4322-7000)/Term 10 (APS4322-5000)/FB Inputs/F{1..9 step 2} Y-Field <-> Data Pointer/HallSensorFieldsXYZ[{76..88 step 3}]  (5 links)
//     Term 9 (APS4322-7000)/Term 10 (APS4322-5000)/FB Inputs/F{1..9 step 2} Z-Field <-> Data Pointer/HallSensorFieldsXYZ[{77..89 step 3}]  (5 links)
//     Term 9 (APS4322-7000)/Term 10 (APS4322-5000)/FB Inputs/G{0..8 step 2} X-Field <-> Data Pointer/HallSensorFieldsXYZ[{90..102 step 3}]  (5 links)
//     Term 9 (APS4322-7000)/Term 10 (APS4322-5000)/FB Inputs/G{0..8 step 2} Y-Field <-> Data Pointer/HallSensorFieldsXYZ[{91..103 step 3}]  (5 links)
//     Term 9 (APS4322-7000)/Term 10 (APS4322-5000)/FB Inputs/G{0..8 step 2} Z-Field <-> Data Pointer/HallSensorFieldsXYZ[{92..104 step 3}]  (5 links)
//     Term 9 (APS4322-7000)/Term 10 (APS4322-5000)/FB Inputs/H{1..9 step 2} X-Field <-> Data Pointer/HallSensorFieldsXYZ[{105..117 step 3}]  (5 links)
//     Term 9 (APS4322-7000)/Term 10 (APS4322-5000)/FB Inputs/H{1..9 step 2} Y-Field <-> Data Pointer/HallSensorFieldsXYZ[{106..118 step 3}]  (5 links)
//     Term 9 (APS4322-7000)/Term 10 (APS4322-5000)/FB Inputs/H{1..9 step 2} Z-Field <-> Data Pointer/HallSensorFieldsXYZ[{107..119 step 3}]  (5 links)
//     Term 9 (APS4322-7000)/Term 10 (APS4322-5000)/FB Inputs/I{0..8 step 2} X-Field <-> Data Pointer/HallSensorFieldsXYZ[{120..132 step 3}]  (5 links)
//     Term 9 (APS4322-7000)/Term 10 (APS4322-5000)/FB Inputs/I{0..8 step 2} Y-Field <-> Data Pointer/HallSensorFieldsXYZ[{121..133 step 3}]  (5 links)
//     Term 9 (APS4322-7000)/Term 10 (APS4322-5000)/FB Inputs/I{0..8 step 2} Z-Field <-> Data Pointer/HallSensorFieldsXYZ[{122..134 step 3}]  (5 links)
//     Term 9 (APS4322-7000)/Term 10 (APS4322-5000)/FB Inputs/J{1..9 step 2} X-Field <-> Data Pointer/HallSensorFieldsXYZ[{135..147 step 3}]  (5 links)
//     Term 9 (APS4322-7000)/Term 10 (APS4322-5000)/FB Inputs/J{1..9 step 2} Y-Field <-> Data Pointer/HallSensorFieldsXYZ[{136..148 step 3}]  (5 links)
//     Term 9 (APS4322-7000)/Term 10 (APS4322-5000)/FB Inputs/J{1..9 step 2} Z-Field <-> Data Pointer/HallSensorFieldsXYZ[{137..149 step 3}]  (5 links)
//     Term 9 (APS4322-7000)/Term 10 (APS4322-5000)/FB Inputs/Status <-> Data Pointer/FeedbackStatus
//   XPlanar MC Project/Axes/0000lckx <-> TcCOM Objects/XPlanar/0000lckx
//     IoToMc/STD <-> OutputsToNC3/HWToNC3
//     McToIo/STD <-> InputsFromNC3/NC3ToHW
//   XPlanar MC Project/Axes/0000lcle <-> TcCOM Objects/XPlanar/0000lcle
//     IoToMc/STD <-> OutputsToNC3/HWToNC3
//     McToIo/STD <-> InputsFromNC3/NC3ToHW
//   DMMS_PLC/DMMS_PLC Instance <-> XPlanar MC Project/Axes/0000lckx
//     PlcTask Inputs/MAIN.fbXMotionUnit.fbXPlanarMover[1].stMoverRef.MCTOPLC/ACT <-> McToPlc/ACT
//     PlcTask Inputs/MAIN.fbXMotionUnit.fbXPlanarMover[1].stMoverRef.MCTOPLC/COORDMODE <-> McToPlc/COORDMODE
//     PlcTask Inputs/MAIN.fbXMotionUnit.fbXPlanarMover[1].stMoverRef.MCTOPLC/SET <-> McToPlc/SET
//     PlcTask Inputs/MAIN.fbXMotionUnit.fbXPlanarMover[1].stMoverRef.MCTOPLC/SETONTRACK <-> McToPlc/SETONTRACK
//     PlcTask Inputs/MAIN.fbXMotionUnit.fbXPlanarMover[1].stMoverRef.MCTOPLC/STD <-> McToPlc/STD
//     PlcTask Outputs/MAIN.fbXMotionUnit.fbXPlanarMover[1].stMoverRef.PLCTOMC/STD <-> PlcToMc/STD
//   DMMS_PLC/DMMS_PLC Instance <-> XPlanar MC Project/Axes/0000lcle
//     PlcTask Inputs/MAIN.fbXMotionUnit.fbXPlanarMover[2].stMoverRef.MCTOPLC/ACT <-> McToPlc/ACT
//     PlcTask Inputs/MAIN.fbXMotionUnit.fbXPlanarMover[2].stMoverRef.MCTOPLC/COORDMODE <-> McToPlc/COORDMODE
//     PlcTask Inputs/MAIN.fbXMotionUnit.fbXPlanarMover[2].stMoverRef.MCTOPLC/SET <-> McToPlc/SET
//     PlcTask Inputs/MAIN.fbXMotionUnit.fbXPlanarMover[2].stMoverRef.MCTOPLC/SETONTRACK <-> McToPlc/SETONTRACK
//     PlcTask Inputs/MAIN.fbXMotionUnit.fbXPlanarMover[2].stMoverRef.MCTOPLC/STD <-> McToPlc/STD
//     PlcTask Outputs/MAIN.fbXMotionUnit.fbXPlanarMover[2].stMoverRef.PLCTOMC/STD <-> PlcToMc/STD
//   DMMS_PLC/DMMS_PLC Instance <-> XPlanar MC Project/Groups/CloseLoopTrack
//     PlcTask Inputs/MAIN.fbXMotionUnit.fbCloseLoopTrack.fbTrackStandard.stTrackRef.MCTOPLC_STD <-> McToPlc/STD
//   DMMS_PLC/DMMS_PLC Instance <-> XPlanar MC Project/Groups/Environment
//     PlcTask Inputs/MAIN.fbXMotionUnit.fbXPlanarSystem.environment.MCTOPLC_STD <-> McToPlc/STD
//   DMMS_PLC/DMMS_PLC Instance <-> XPlanar MC Project/Groups/PipetteBufferConTrack
//     PlcTask Inputs/MAIN.fbXMotionUnit.fbTrackPipetteBufferCon.fbTrackStandard.stTrackRef.MCTOPLC_STD <-> McToPlc/STD
//   DMMS_PLC/DMMS_PLC Instance <-> XPlanar MC Project/Groups/PipettePostBufferTrack
//     PlcTask Inputs/MAIN.fbXMotionUnit.fbTrackPipettePostBuffer.fbTrackStandard.stTrackRef.MCTOPLC_STD <-> McToPlc/STD
//   DMMS_PLC/DMMS_PLC Instance <-> XPlanar MC Project/Groups/PipettePreBufferTrack
//     PlcTask Inputs/MAIN.fbXMotionUnit.fbTrackPipettePreBuffer.fbTrackStandard.stTrackRef.MCTOPLC_STD <-> McToPlc/STD
//   DMMS_PLC/DMMS_PLC Instance <-> XPlanar MC Project/Groups/PipetteTrack
//     PlcTask Inputs/MAIN.fbXMotionUnit.fbTrackPipette.fbTrackStandard.stTrackRef.MCTOPLC_STD <-> McToPlc/STD
//   DMMS_PLC/DMMS_PLC Instance <-> XPlanar MC Project/Groups/PuncherBufferTrack
//     PlcTask Inputs/MAIN.fbXMotionUnit.fbTrackBufferPuncher.fbTrackStandard.stTrackRef.MCTOPLC_STD <-> McToPlc/STD
//   DMMS_PLC/DMMS_PLC Instance <-> XPlanar MC Project/Groups/PuncherSeperateTrack
//     PlcTask Inputs/MAIN.fbXMotionUnit.fbPuncherSeperate.fbTrackStandard.stTrackRef.MCTOPLC_STD <-> McToPlc/STD
//   DMMS_PLC/DMMS_PLC Instance <-> XPlanar MC Project/Groups/PuncherWellplateTrack
//     PlcTask Inputs/MAIN.fbXMotionUnit.fbTrackPuncherWellplate.fbTrackStandard.stTrackRef.MCTOPLC_STD <-> McToPlc/STD
//   DMMS_PLC/DMMS_PLC Instance <-> XPlanar MC Project/Groups/StradeFirstSegTrack
//     PlcTask Inputs/MAIN.fbXMotionUnit.fbTrackStradeFirstSeg.fbTrackStandard.stTrackRef.MCTOPLC_STD <-> McToPlc/STD
//   DMMS_PLC/DMMS_PLC Instance <-> XPlanar MC Project/Groups/StradeSecondSegTrack
//     PlcTask Inputs/MAIN.fbXMotionUnit.fbTrackStradeSecondSeg.fbTrackStandard.stTrackRef.MCTOPLC_STD <-> McToPlc/STD
//   DMMS_PLC/DMMS_PLC Instance <-> XPlanar MC Project/Groups/UserInteractionTrack
//     PlcTask Inputs/MAIN.fbXMotionUnit.fbTrackUserInteraction.fbTrackStandard.stTrackRef.MCTOPLC_STD <-> McToPlc/STD
//   DMMS_PLC/DMMS_PLC Instance <-> XPlanar MC Project/Groups/XPlanar
//     PlcTask Inputs/MAIN.fbXMotionUnit.fbXPlanarSystem.group.MCTOPLC_STD <-> McToPlc/STD

CONFIGURATION DMMS_PLC
    RESOURCE PLC ON TwinCAT3
        TASK PlcTask(INTERVAL := T#10ms, PRIORITY := 20);
        PROGRAM MAIN WITH PlcTask : MAIN;
    END_RESOURCE
END_CONFIGURATION

// ---- DUTs/Communiction/Movers/ST_ComOut_ExportMover.TcDUT
{attribute 'pack_mode' := '1'}  // needed for python pyads reading
TYPE ST_ComOut_ExportMover :
STRUCT
	Avaiable: BOOL; 
	Error: BOOL;
	CurrentTaskFinished:BOOL;
	Status_Word: INT; 
	Error_ID: INT;
	MoverType:INT;
	CurrentStation: UINT;
	LastTask: UDINT; 
	CurrentTask: UDINT; 
	TrackID: UDINT;
	TrackPos: LREAL;
	Id: STRING(13);
	Position : MoverPositionUnion;
	
	
END_STRUCT
END_TYPE

// ---- DUTs/Communiction/Station/ST_Com_ExportStation.TcDUT
TYPE ST_Com_ExportStation :
STRUCT
		IN: 		ST_ComIn_ExportStation;
		OUT:		ST_ComOut_ExportStation;
END_STRUCT
END_TYPE

// ---- Mover/DUTs/MoverPositionUnion.TcDUT
{attribute 'pack_mode' := '1'}
TYPE MoverPositionUnion :
	UNION
		arr: ARRAY[1..6] OF LREAL;
		vec: MoverVector;
	END_UNION
END_TYPE

// ---- Mover/DUTs/ST_ManMov_FreeMove.TcDUT
{attribute 'pack_mode' := '1'}  // needed for python pyads reading
TYPE ST_ManMov_FreeMove :
STRUCT
	move_position_CMD_enable:BOOL;
	move_position_CMD_done: BOOL;
	move_position :MoverVector;
END_STRUCT
END_TYPE

// ---- Mover/DUTs/ST_ProcessResult.TcDUT
{attribute 'pack_mode' := '1'}  // needed for python pyads reading
TYPE ST_ProcessResult :
STRUCT
	
	Done:BOOL;
	OK:BOOL;
	Damage:BOOL;
	NOK:BOOL;
	NOK_Resaon: INT;
	
END_STRUCT
END_TYPE

// ---- Stations/DUTs/ST_StationReturn.TcDUT
TYPE ST_StationReturn :
STRUCT
	Done	: BOOL;
	stState	: INT;
END_STRUCT
END_TYPE

// ---- Mover/I_MoverApplication.TcIO
INTERFACE I_MoverApplication

METHOD Cycle
END_METHOD

METHOD ManualMovement : BOOL
VAR_INPUT
	bReset: bool;
END_VAR
END_METHOD

PROPERTY P_ControlData : Reference to ST_ControlData
GET
END_GET
SET
END_SET
END_PROPERTY

PROPERTY P_MoverConfiguration : Reference to  ST_MoverConfiguration
GET
END_GET
SET
END_SET
END_PROPERTY

PROPERTY P_MoverID : STRING
GET
END_GET
SET
END_SET
END_PROPERTY

PROPERTY P_MoverIndex : INT
GET
END_GET
SET
END_SET
END_PROPERTY

PROPERTY P_ProcessTask :  ST_ProcessTask
GET
END_GET
SET
END_SET
END_PROPERTY

PROPERTY P_ProductData : Reference to ST_ProductData
GET
END_GET
SET
END_SET
END_PROPERTY

PROPERTY P_TrackId : UDINT
GET
END_GET
SET
END_SET
END_PROPERTY

PROPERTY std : I_XPlanarMoverStandard
GET
END_GET
SET
END_SET
END_PROPERTY

END_INTERFACE

// ---- Stations/Base/I_Station.TcIO
INTERFACE I_Station

METHOD Clear : BOOL
VAR_INPUT
END_VAR
END_METHOD

METHOD Cycle : BOOL
VAR_INPUT
END_VAR
END_METHOD

METHOD Init : BOOL
END_METHOD

PROPERTY P_bInitDone : BOOL
GET
END_GET
END_PROPERTY

PROPERTY P_eProcessMode : E_ProcessMode
GET
END_GET
SET
END_SET
END_PROPERTY

PROPERTY P_List_Station : I_List
GET
END_GET
END_PROPERTY

PROPERTY P_List_Switch_Input_E : I_List
GET
END_GET
END_PROPERTY

PROPERTY P_List_Switch_Input_N : I_List
GET
END_GET
END_PROPERTY

PROPERTY P_List_Switch_Input_S : I_List
GET
END_GET
END_PROPERTY

PROPERTY P_List_Switch_Input_W : I_List
GET
END_GET
END_PROPERTY

PROPERTY P_nErrorCode : UDINT
GET
END_GET
END_PROPERTY

PROPERTY P_Position : ST_StationPosition
GET
END_GET
END_PROPERTY

PROPERTY P_ProcessClearance : DINT
GET
END_GET
END_PROPERTY

PROPERTY P_ProcessRequest : UDINT
GET
END_GET
SET
END_SET
END_PROPERTY

PROPERTY P_ProcessState : DINT
GET
END_GET
END_PROPERTY

PROPERTY P_StationTaskList : array[1..200] of UDINT
GET
END_GET
SET
END_SET
END_PROPERTY

METHOD Process : BOOL
END_METHOD

END_INTERFACE

// ---- Mover/FB_ApplicationMover.TcPOU
FUNCTION_BLOCK FB_ApplicationMover IMPLEMENTS I_MoverApplication
VAR
	ipMoverStandard	: I_XPlanarMoverStandard;
	
	stProductData	: ST_ProductData;
	eMoverType 		: ST_EMoverLoadType;
	
	nMoverIndex		: INT;
	sMoverID 		: STRING(13) := '00001111';
	
	nTrackId		: UDINT;
	
	// customer Data
	bIsLoaded		: BOOL;	
	stControlData	:ST_ControlData;
	stMoverConfiguration: ST_MoverConfiguration;
	stProcessTask: St_ProcessTask;
	
	
				
END_VAR

METHOD Cycle


VAR_INST
	nTestCounter	: UINT;
	index: UDINT;
	
END_VAR
IF std <> 0 THEN

	std.cycle();
		
		// comunication data 
		
	IF communication.RunAplicationComm THEN 
		FOR index:=1 TO GVL.gc_nMaxNumberMovers DO 
			
			IF communication.g_Com_Movers[index].IN.id= THIS^.P_MoverID THEN 
				
				Communication.g_Com_Movers[index].OUT.Id:=THIS^.P_MoverID;
				Communication.g_Com_Movers[index].OUT.TrackID:=THIS^.P_TrackId;
				
			IF communication.g_Com_Movers[index].IN.MoverType=1 THEN 
				eMoverType :=ST_EMoverLoadType.Wellplate ;
			ELSIF communication.g_Com_Movers[index].IN.MoverType=2 THEN 
				eMoverType :=ST_EMoverLoadType.Gripper ;
			ELSIF communication.g_Com_Movers[index].IN.MoverType=3 THEN 
				eMoverType :=ST_EMoverLoadType.PipetteTips ;
			END_IF	
				
				//Position 
				Communication.g_Com_Movers[index].OUT.Avaiable:=(THIS^.std.P_State=3);
				Communication.g_Com_Movers[index].OUT.position.vec := THIS^.std.P_ActPosition;
	
				Communication.g_Com_Movers[index].OUT.Position.vec.x:=THIS^.std.P_ActPosition.x;
				Communication.g_Com_Movers[index].OUT.Position.vec.y:=THIS^.std.P_ActPosition.y;
				Communication.g_Com_Movers[index].OUT.Position.vec.c:=THIS^.std.P_ActPosition.c;
				
				//configuration
				stMoverConfiguration.MoverType:= Communication.g_Com_Movers[index].IN.MoverType;
				communication.g_Com_Movers[index].out.MoverType:= THIS^.stMoverConfiguration.MoverType;
	
				stMoverConfiguration.WellplateData:=Communication.g_Com_Movers[index].IN.WellplateData;
				
				//ControlData
				stControlData.StatusWord:= THIS^.std.P_State;
				Communication.g_Com_Movers[index].OUT.Status_Word:= stControlData.StatusWord;
				stControlData.ControlWord:= communication.g_Com_Movers[index].IN.ControlWord;
				
				//Process Task 
				Communication.g_Com_Movers[index].OUT.LastTask:= stProcessTask.LastTask;
				Communication.g_Com_Movers[index].OUT.CurrentTask:= stProcessTask.CurrentTask;
				Communication.g_Com_Movers[index].OUT.CurrentTaskFinished:= stProcessTask.CurrentTaskFinished;
				stProcessTask.TaskToProcessed:=Communication.g_Com_Movers[index].IN.TaskToProcessed;
			
				
		
					IF Communication.g_Com_Movers[index].IN.Reset THEN
						
						ipMoverStandard.Reset(slogMessage:='mover reset');
						
					END_IF

			
			
			
			END_IF
		END_FOR
	END_IF
	
	
END_IF
END_METHOD

METHOD ManualMovement : BOOL
VAR_INPUT
	bReset: bool;
END_VAR

VAR_INST
	nTestCounter	: UINT;
	index: UDINT;
	Com_Index: UDINT;
	nMovementSequence : UDINT;
	
	
END_VAR

VAR
	ManMovements: 	ST_ManualMovements;
	targetPos 						:  PositionXYC;
	fTargetPosOnTrack 				: LREAL;
	stOptionsJoinTrack				: ST_JoinTrackOptions;
	stMoveOnTrackOptions			: ST_MoveOnTrackOptions;
	stMoveToPositionOptions			: ST_MoveToPositionOptions;
	bMoversJoined 					: BOOL;
	bMoverError						: BOOL;
	bMoversInPos					: BOOL;
	strInfo							: STRING;
	
END_VAR
	IF communication.RunAplicationComm THEN 
		FOR index:=1 TO GVL.gc_nMaxNumberMovers DO 
			
			IF communication.g_Com_Movers[index].IN.id= THIS^.P_MoverID THEN
				
				ManMovements:= communication.g_Com_Movers[index].ManualMovements;
				Com_Index:=index;
				
			END_IF
			
		END_FOR
		
	END_IF
	
	
	
	IF bReset OR  Communication.g_Com_GlobalState.IN.Stop   OR Communication.g_Com_GlobalState.IN.Reset THEN 
	ManualMovement := FALSE;
	nMovementSequence := 0;
END_IF

CASE nMovementSequence OF
	

0: //init
		
 	// wait for enabling  process 
			 IF Communication.g_Com_GlobalState.IN.Start AND NOT Communication.g_Com_GlobalState.IN.EOC_Stop  AND Com_Index <>0 THEN 
				IF Communication.g_Com_GlobalState.IN.ProgramType =2 THEN 
					  nMovementSequence := 100;
				
					   ELSIF Communication.g_Com_GlobalState.IN.ProgramType =3 THEN 
					  nMovementSequence := 200;
				END_IF								
					 
			 END_IF
			 




100:	 // position test 
	
		// leave track
		IF ipMoverStandard.P_CommandMode= MC_PLANAR_MOVER_COMMAND_MODE.OnTrack AND  NOT ipMoverStandard.P_Busy THEN

			ipMoverStandard.LeaveTrackInPosition( strInfo, FALSE);
			nMovementSequence := nMovementSequence +1;
		ELSE 
			nMovementSequence := 110;
		END_IF


101:
			IF ipMoverStandard.P_LeaveTrackInPosition.Done THEN
				P_TrackId:=0;
				nMovementSequence := 110;
			ELSIF ipMoverStandard.P_LeaveTrackInPosition.Error THEN
				nMovementSequence := nMovementSequence +4;
			END_IF	
				


110://setup state 
		IF NOT ManMovements.FreeMove.move_position_CMD_enable THEN 
				ManMovements.FreeMove.move_position_CMD_done:= FALSE;
				communication.g_Com_Movers[Com_Index].ManualMovements:=ManMovements;
		END_IF
						nMovementSequence := nMovementSequence +  1;					  
				
111: 	//execute command 
stMoveToPositionOptions.useOrientation:= TRUE;
	targetPos.x:=	ManMovements.FreeMove.move_position.x ;
	targetPos.y:=	ManMovements.FreeMove.move_position.y;
	targetPos.C:=	ManMovements.FreeMove.move_position.C;
					 // targetpos.ShiftByXy(ManMovements.move_position.x,ManMovements.move_position.y);
				
	


			IF  ManMovements.FreeMove.move_position_CMD_enable AND NOT ManMovements.FreeMove.move_position_CMD_done  THEN 
					ipMoverStandard.MoveToPositionEXt('move to XY', targetPos, 100, 2500, 2500, 25000,stMoveToPositionOptions);
					nMovementSequence := nMovementSequence +  1;
			ELSE
				nMovementSequence := 0;
			END_IF
				
		
	
	
112: 	// check commad result 

		
		IF ipMoverStandard.P_MoveToPositionExt.Done THEN
			ManMovements.FreeMove.move_position_CMD_done:= TRUE;
			communication.g_Com_Movers[Com_Index].ManualMovements:=ManMovements;
			nMovementSequence :=  0;
		ELSIF ipMoverStandard.P_MoveToPositionExt.Error THEN
			nMovementSequence := nMovementSequence +  3;
		END_IF				
		
		
200:
		 IF NOT ManMovements.MoveTrack.move_track_CMD_done THEN 
				IF ManMovements.MoveTrack.join_track AND ManMovements.MoveTrack.move_track_no<>0 THEN 
					nMovementSequence := 210;
				ELSIF ManMovements.MoveTrack.leave_track THEN
					nMovementSequence := 220;
				ELSIF ManMovements.MoveTrack.move_track AND ManMovements.MoveTrack.move_track_no<>0 THEN 
					nMovementSequence := 230;
				ELSE
					nMovementSequence := 0;
				END_IF
		END_IF
		
		IF NOT ManMovements.MoveTrack.move_track_CMD_enable THEN 
			ManMovements.MoveTrack.move_track_CMD_done := FALSE;
			communication.g_Com_Movers[Com_Index].ManualMovements:=ManMovements;
		END_IF

210:	
		stOptionsJoinTrack.useOrientation := TRUE;
	
		IF (ipMoverStandard.P_CommandMode<> MC_PLANAR_MOVER_COMMAND_MODE.OnTrack OR  INT_TO_UDINT(ManMovements.MoveTrack.move_track_no)<>P_TrackId)
			AND NOT ipMoverStandard.P_Busy
			AND ManMovements.MoveTrack.move_track_CMD_enable THEN
			ipMoverStandard.JoinTrack('Joining track', GVL.g_Tracks[ManMovements.MoveTrack.move_track_no].std, 250, 1250, 12500, stOptionsJoinTrack);
				nMovementSequence := nMovementSequence + 1;
			ELSE 
				nMovementSequence := 0;
		END_IF
	
	
		
211:
	
			bMoversJoined := ipMoverStandard.P_JoinTrack.Done;
			bMoverError :=  ipMoverStandard.P_JoinTrack.Error;			
		
	IF bMoversJoined THEN
		ManMovements.MoveTrack.move_track_CMD_done:=TRUE;
		communication.g_Com_Movers[Com_Index].ManualMovements:=ManMovements;
		P_TrackId:=INT_TO_UDINT(ManMovements.MoveTrack.move_track_no);
		nMovementSequence := 0;
	ELSIF bMoverError THEN
 			nMovementSequence := nMovementSequence + 4;
	END_IF

		
	
		
220:
		
		IF ipMoverStandard.P_CommandMode= MC_PLANAR_MOVER_COMMAND_MODE.OnTrack AND  NOT ipMoverStandard.P_Busy AND ManMovements.MoveTrack.move_track_CMD_enable  THEN

			ipMoverStandard.LeaveTrackInPosition( strInfo, FALSE);
			nMovementSequence := nMovementSequence +1;
		ELSE 
			nMovementSequence := 0;
		END_IF


221:
			IF ipMoverStandard.P_LeaveTrackInPosition.Done THEN
				ManMovements.MoveTrack.move_track_CMD_done:=TRUE;
				communication.g_Com_Movers[Com_Index].ManualMovements:=ManMovements;
				P_TrackId:=0;
				nMovementSequence := 0;
			ELSIF ipMoverStandard.P_LeaveTrackInPosition.Error THEN
				nMovementSequence := nMovementSequence +4;
			END_IF	
			
230:

		
		stMoveOnTrackOptions.gap := 120;
		fTargetPosOnTrack:=ManMovements.MoveTrack.move_track_position;
		stMoveOnTrackOptions.dynamicMode := MC_DYNAMICS_REDUCTION_MODE.AccelerationLimitedVelocity;
		stMoveOnTrackOptions.direction := MC_DIRECTION.mcDirectionShortestWay;
		IF   NOT ipMoverStandard.P_Busy AND ManMovements.MoveTrack.move_track_CMD_enable  THEN
				 ipMoverStandard.MoveOnTrackEXT('move on track', GVL.g_Tracks[ManMovements.MoveTrack.move_track_no].std, fTargetPosOnTrack,
								300, 3000, 15000, stMoveOnTrackOptions);
				nMovementSequence := nMovementSequence +1;
		 END_IF
		 


	231:
			bMoversInPos :=  ipMoverStandard.P_MoveOnTrackExt.Done;
			bMoverError := ipMoverStandard.P_MoveOnTrackExt.Error;
	
		
		IF bMoversInPos THEN
			ManMovements.MoveTrack.move_track_CMD_done:=TRUE;
			communication.g_Com_Movers[Com_Index].ManualMovements:=ManMovements;
			nMovementSequence := 0;
		ELSIF bMoverError THEN
			nMovementSequence := nMovementSequence +  3;
		END_IF
			
			
			
	END_CASE
END_METHOD

PROPERTY P_ControlData : Reference to ST_ControlData
GET
P_ControlData := stControlData;
END_GET
SET
stControlData := P_ControlData;
END_SET
END_PROPERTY

PROPERTY P_MoverConfiguration : Reference to  ST_MoverConfiguration
GET
P_MoverConfiguration := stMoverConfiguration;
END_GET
SET
stMoverConfiguration := P_MoverConfiguration;
END_SET
END_PROPERTY

PROPERTY P_MoverID : STRING
GET
P_MoverID := sMoverID;
END_GET
SET
sMoverID := P_MoverID;
END_SET
END_PROPERTY

PROPERTY P_MoverIndex : INT
GET
P_MoverIndex := nMoverIndex;
END_GET
SET
nMoverIndex := P_MoverIndex;
END_SET
END_PROPERTY

PROPERTY P_ProcessTask : ST_ProcessTask
GET
P_ProcessTask := stProcessTask;
END_GET
SET
stProcessTask := P_ProcessTask;
END_SET
END_PROPERTY

PROPERTY P_ProductData : Reference to ST_ProductData
GET
P_ProductData REF= stProductData;
END_GET
SET
stProductData := P_ProductData;
END_SET
END_PROPERTY

PROPERTY P_TrackId : UDINT
GET
P_TrackId := nTrackId;
END_GET
SET
nTrackId := P_TrackId;
END_SET
END_PROPERTY

PROPERTY std : I_XPlanarMoverStandard
GET
IF ipMoverStandard <> 0 THEN
	std := ipMoverStandard;	
END_IF
END_GET
SET
ipMoverStandard := std;
END_SET
END_PROPERTY

END_FUNCTION_BLOCK

// ---- POUs/FB_MotionSystem.TcPOU
FUNCTION_BLOCK FB_MotionSystem
VAR_INPUT
END_VAR
VAR_OUTPUT
END_VAR
VAR
	fbXPlanarSystem	: FB_XPlanarSystem;
	stMoverDetectionInfos   : ST_TcIoMoverDetectionInfos;
	fbTcIoXPlanarEnv	:FB_TcIoXPlanarEnvironment  ; 
	ipXpu	: I_TcIoXPlanarProcessingUnit;

	
	fbMover					: ARRAY [1..GVL.gc_nMaxNumberMovers] OF FB_ApplicationMover;
	fbXPlanarMover : ARRAY [1..GVL.gc_nMaxNumberMovers] OF FB_XPlanarMoverStandard; 
	
	nStartupSequence : UDINT;
	nStartingSequence : UDINT;
	nExecutingSequence : UDINT;
	nResettingSequence 	: UDINT;
	nRecoverySequence : UDINT;
	
	// Helper
	bDone 					: BOOL;
	idx						: UDINT;
	nForCounter 			: UDINT;	
	nErrorID				: UDINT;
	bMoverError				: BOOL;	
	
	// TRACKS
	fbTrackPuncherWellplate		: FB_PuncherWellplateTrack;
	fbTrackBufferPuncher		: FB_PuncherBufferTrack;
	fbPuncherSeperate			: FB_PuncherSeperateTrack;
	fbTrackStradeFirstSeg		: FB_StradeFirstSegTrack;
	fbTrackStradeSecondSeg		: FB_StradeSecondSegTrack;
	fbTrackPipettePreBuffer		: FB_PipettePreBufferTrack;
	fbTrackPipette				: FB_PipetteTrack;
	fbTrackPipettePostBuffer	: FB_PipettePostBufferTrack;
	fbTrackPipetteBufferCon		: FB_PipetteBufferConTrack;
	fbTrackUserInteraction		: FB_UserInteractionTrack;
	fbCloseLoopTrack			: FB_CloseLoopTrack;

	
	// STATIONS
	fbPuncherStation : FB_PuncherStation;
	fbPuncherSeparateStation : FB_PuncherSeparateStation;
	fbPuncherBufferStation : FB_PuncherBufferStation;
	
	bAssignmentComplete 		: BOOL;
	

	
END_VAR

METHOD Cycle
VAR_INPUT
END_VAR

VAR
	index	: UDINT;
END_VAR

fbXPlanarSystem.Cycle();

IF bAssignmentComplete THEN

	FOR index := 1 TO  MoverCount DO
		fbXPlanarMover[index].Cycle();
		GVL.g_Movers[index].Cycle();
		fbMover[index].Cycle();
	END_FOR

	FOR index := 1 TO GVL.gc_NumberTracks DO
		GVL.g_Tracks[index].Cycle();
	END_FOR	
END_IF
END_METHOD

METHOD Execute : BOOL
VAR_INPUT
	bReset : BOOL;
END_VAR

VAR
	index : UDINT;
	com_index:UDINT;
	stMoveOnTrackOptions: ST_MoveOnTrackOptions;
END_VAR

VAR_INST
	
	stOptionsJoinTrack				: ST_JoinTrackOptions;
	bMoversJoined 					: BOOL;
	nMoverToTurnBack				: UDINT;
	nTrackToCheck					:UDINT; 
	nDistanceToTrack				:LREAL;
	nDistanceToTargetTrack			: ARRAY[1..moverCount] OF REAL;
	nTargetTrack					: ARRAY[1..moverCount] OF UDINT;
	bMoversinPos					:BOOL;
	bMoverError						:BOOL;
	
	
END_VAR
IF bReset OR  Communication.g_Com_GlobalState.IN.EOC_Stop   THEN
	Execute := FALSE;
	nExecutingSequence := 0;
END_IF

CASE nExecutingSequence OF
	

0: //init
		bMoversinPos := FALSE;
		bMoverError := FALSE;
 	// wait for enabling  process 
			 IF Communication.g_Com_GlobalState.IN.Start AND NOT Communication.g_Com_GlobalState.IN.EOC_Stop THEN 
				 IF Communication.g_Com_GlobalState.IN.ProgramType =1 THEN 
				 nExecutingSequence := 10;
			
				 Communication.g_Com_GlobalState.OUT.ProgramType:=1;
				 
				 ELSIF Communication.g_Com_GlobalState.IN.ProgramType =2 THEN 
					  nExecutingSequence := 20;
					   Communication.g_Com_GlobalState.OUT.InCycle:=FALSE; 
						Communication.g_Com_GlobalState.OUT.ProgramType:=2;
				
					   ELSIF Communication.g_Com_GlobalState.IN.ProgramType =3 THEN 
					  nExecutingSequence := 30;
					  	Communication.g_Com_GlobalState.OUT.InCycle:=FALSE; 
						Communication.g_Com_GlobalState.OUT.ProgramType:=3;
						
				END_IF								
					 
			 END_IF
			 

			 
10:			 // auto cycle 
			// check all movers join to track
			
			FOR index := 1 TO gvl. g_nMoverCount DO
			IF fbXPlanarMover[index].P_CommandMode<> MC_PLANAR_MOVER_COMMAND_MODE.OnTrack THEN 
				
					nExecutingSequence := nExecutingSequence + 1;
					index:=nMoverToTurnBack;
				RETURN ;
			END_IF
			END_FOR 
			nExecutingSequence := nExecutingSequence + 5;
	
11: // look for for nearest track 
	
	
//	FOR nMoverToTurnBack := 1 TO  gvl.g_nMoverCount DO
		nDistanceToTargetTrack[nMoverToTurnBack]:= 999999;
		
		FOR nTrackToCheck :=1 TO GVL.gc_NumberTracks DO 
		nDistanceToTrack := fbXPlanarMover[ nMoverToTurnBack].GetDistanceToTrack(GVL.g_Tracks[nTrackToCheck].std);
		
		IF nDistanceToTrack < nDistanceToTargetTrack[nMoverToTurnBack] AND nDistanceToTrack<> -1 THEN 
			nDistanceToTargetTrack[nMoverToTurnBack]:=nDistanceToTrack;
			nTargetTrack[nMoverToTurnBack] :=nTrackToCheck;
		END_IF
		
	END_FOR
	
	//END_FOR
	
	nRecoverySequence := nRecoverySequence +10;
	
12: // join to track

		stOptionsJoinTrack.useOrientation := TRUE;
		
		//FOR index := 1 TO gvl.g_nMoverCount DO
		
		IF fbXPlanarMover[nMoverToTurnBack].P_CommandMode<> MC_PLANAR_MOVER_COMMAND_MODE.OnTrack THEN
			IF  GVL.g_Movers[nMoverToTurnBack].P_MoverConfiguration.MoverType= ST_EMoverLoadType.Wellplate THEN 

				fbXPlanarMover[nMoverToTurnBack].JoinTrack('Joining track', GVL.g_Tracks[nTargetTrack[nMoverToTurnBack]].std, 250, 1250, 12500, stOptionsJoinTrack);
			
			ELSIF  GVL.g_Movers[nMoverToTurnBack].P_MoverConfiguration.MoverType= ST_EMoverLoadType.Gripper THEN 
					
				fbXPlanarMover[nMoverToTurnBack].JoinTrack('Joining track', GVL.g_Tracks[11].std, 250, 1250, 12500, stOptionsJoinTrack);
			
			ELSIF  GVL.g_Movers[nMoverToTurnBack].P_MoverConfiguration.MoverType= ST_EMoverLoadType.PipetteTips THEN 
					
				fbXPlanarMover[nMoverToTurnBack].JoinTrack('Joining track', GVL.g_Tracks[7].std, 250, 1250, 12500, stOptionsJoinTrack);
			
			END_IF
		END_IF
		
			
		//END_FOR
	
		nRecoverySequence := nRecoverySequence + 1;
		
	13:
		bMoversJoined := TRUE;
		bMoverError := FALSE;
		//FOR index := 1 TO moverCount DO
			
			bMoversJoined := bMoversJoined AND fbXPlanarMover[nMoverToTurnBack].P_JoinTrack.Done;
			IF  fbXPlanarMover[nMoverToTurnBack].P_JoinTrack.Done THEN 
				gvl.g_Movers[nMoverToTurnBack].P_TrackId:=nTargetTrack[nMoverToTurnBack];
			END_IF
			bMoverError := bMoverError OR fbXPlanarMover[nMoverToTurnBack].P_JoinTrack.Error;	
			 	
	//	END_FOR
		
	IF bMoversJoined THEN
			nRecoverySequence := 10;
	ELSIF bMoverError THEN
 			nRecoverySequence := nRecoverySequence + 4;
	END_IF
			
14: 	//send mover to station 
	  	  
		FOR index := 1 TO gvl.g_nMoverCount DO
			 IF fbXPlanarMover[index].P_TrackId= GVL.TrackPuncherWellplate 
			AND GVL.g_Movers[index].P_MoverConfiguration.MoverType= ST_EMoverLoadType.Wellplate
			
			  THEN 
				 fbPuncherStation.P_List_Switch_Input_W.AddMover(GVL.g_Movers[index].std);
			 END_IF

			  IF GVL.g_Movers[index].P_MoverConfiguration.MoverType= ST_EMoverLoadType.Gripper THEN 
				 fbPuncherSeparateStation.P_List_Switch_Input_N.AddMover(GVL.g_Movers[index].std);
			  END_IF
			  
			 
		END_FOR

	
			nExecutingSequence := nExecutingSequence+1;

15: 		// set process mode 
		 	 FOR index := 1 TO GVL.gc_NumberStations DO
 			GVL.g_Stations[index].P_eProcessMode := E_ProcessMode.Production;		   
	 	   END_FOR
			
				nExecutingSequence := nExecutingSequence+1;

16:			//process method
			Communication.g_Com_GlobalState.OUT.InCycle:=TRUE; 
			fbPuncherStation.Process();
			fbPuncherSeparateStation.Process();
			
			nExecutingSequence := 0;

20,30: 

		 	 FOR index := 1 TO GVL.gc_NumberStations DO
 			GVL.g_Stations[index].P_eProcessMode := E_ProcessMode.None;		   
	 	   END_FOR
	

		FOR index := 1 TO gvl. g_nMoverCount DO
		
		GVL.g_Movers[index].ManualMovement(FALSE);
		END_FOR

	nExecutingSequence := 0;

// test movement

	
// 	 FOR index := 1 TO GVL.gc_NumberStations DO
// 			GVL.g_Stations[index].P_eProcessMode := E_ProcessMode.Production;		   
// 	   END_FOR
// 		
// 	 
// 
// 	nExecutingSequence := nExecutingSequence +10;
// 
// 	10:
// 	  
// 	   
//   IF fbXPlanarMover[nTestID].P_Enable.Done THEN 
// 		stMoveOnTrackOptions.gap := 120;
// 		stMoveOnTrackOptions.direction := MC_DIRECTION.mcDirectionShortestWay;
// 		stMoveOnTrackOptions.dynamicMode := MC_DYNAMICS_REDUCTION_MODE.AccelerationLimitedVelocity;
// 
// 					
// 				fTargetPosOnTrack[1]:= GVL.g_Tracks[9].P_TrackLength;			
// 				fbXPlanarMover[nTestID].MoveOnTrackExt('move on track', GVL.g_Tracks[9].std, fTargetPosOnTrack[1],
// 								500, 2500, 50000, stMoveOnTrackOptions);
// 		nExecutingSequence := nExecutingSequence +1;
// 		 
// 	END_IF
// 
// 	11:
// 		bMoversInPos := TRUE;
// 		bMoverError := FALSE;
// 		
// 		
// 			bMoversInPos := bMoversInPos AND fbXPlanarMover[nTestID].P_MoveOnTrackExt.Done;
// 			bMoverError := bMoverError OR fbXPlanarMover[nTestID].P_MoveOnTrackExt.Error;
// 	
// 		
// 		IF bMoversInPos THEN
// 			nExecutingSequence := nExecutingSequence + 9;
// 		ELSIF bMoverError THEN
// 			nExecutingSequence := nExecutingSequence +  4;
// 		END_IF
// 
// 	20:
// 		FOR nForCounter:=1 TO GVL.gc_NumberStations DO
// 		IF GVL.g_Stations[nForCounter] <> 0 THEN
// 			GVL.g_Stations[nForCounter].Process();
// 			
// 			IF GVL.g_Stations[nForCounter].P_nErrorCode > 0 THEN
// 				nProcessFeedback := GVL.g_Stations[nForCounter].P_nErrorCode;
// 			END_IF
// 		END_IF
// 	END_FOR	
// 		nExecutingSequence := nExecutingSequence +10;
// 		
// 	30:
// 		stMoveOnTrackOptions.gap := 120;
// 		stMoveOnTrackOptions.direction := MC_DIRECTION.mcDirectionShortestWay;
// 		stMoveOnTrackOptions.dynamicMode := MC_DYNAMICS_REDUCTION_MODE.AccelerationLimitedVelocity;
// 		
// 		fTargetPosOnTrack[1] := GVL.g_Tracks[7].P_TrackLength;;
// 		fbXPlanarMover[nTestID].MoveOnTrackExt('move on track', GVL.g_Tracks[7].std, fTargetPosOnTrack[1],
// 												500, 2500, 50000, stMoveOnTrackOptions
// 		);
// 		nExecutingSequence := nExecutingSequence +1;
// 	31:
// 		// Movers moving on track
// 			bMoversInPos := TRUE;
// 			bMoverError := FALSE;
// 		
// 					bMoversInPos := bMoversInPos AND	fbXPlanarMover[nTestID].P_MoveOnTrackExt.Done;
// 					bMoverError := bMoverError OR fbXPlanarMover[nTestID].P_MoveOnTrackExt.Error;
// 	
// 			IF bMoversInPos THEN
// 			nExecutingSequence := nExecutingSequence + 9;
// 			ELSIF bMoverError THEN
// 			nExecutingSequence := nExecutingSequence + 4;
// 			END_IF
// 
// 
// 	40: 
// 
// 		stMoveOnTrackOptions.gap := 120;
// 		stMoveOnTrackOptions.direction := MC_DIRECTION.mcDirectionShortestWay;
// 		stMoveOnTrackOptions.dynamicMode := MC_DYNAMICS_REDUCTION_MODE.AccelerationLimitedVelocity;
// 		
// 		fTargetPosOnTrack[1] := GVL.g_Tracks[8].P_TrackLength;;
// 		fbXPlanarMover[nTestID].MoveOnTrackExt('move on track', GVL.g_Tracks[8].std, fTargetPosOnTrack[1],
// 												500, 2500, 50000, stMoveOnTrackOptions	);									
// 												
// 												
// 		nExecutingSequence := nExecutingSequence +1;
// 	41:
// 		// Movers moving on track
// 			bMoversInPos := TRUE;
// 			bMoverError := FALSE;
// 		
// 					bMoversInPos := bMoversInPos AND	fbXPlanarMover[nTestID].P_MoveOnTrackExt.Done;
// 					bMoverError := bMoverError OR fbXPlanarMover[nTestID].P_MoveOnTrackExt.Error;
// 	
// 			IF bMoversInPos THEN
// 			nExecutingSequence := nExecutingSequence + 9;
// 			ELSIF bMoverError THEN
// 			nExecutingSequence := nExecutingSequence + 4;
// 			END_IF
// 	
// 	
// 
// 	50:
// 		Execute := FALSE; // must be aborted manually
// 		nExecutingSequence := 0; // endless loop
	
END_CASE
END_METHOD

METHOD MoverPreparation : BOOL
VAR_INPUT
	bReset 	: BOOL;
END_VAR


VAR_INST
	
	nStatePreparation		: DINT;
	
	
	operationMode				: XPlanarOperationMode; 
	
	idx2						: UDINT;

	nTileDcLinkVoltage			: LREAL;
	bTilePowerOK				: BOOL;
	bTilePowerOverview			: ARRAY[1..GVL.gc_MaxNumberTiles] OF BOOL;
	bPowerOK					: BOOL;
	bPowerMissing				: BOOL;
	nTileCount					: UDINT;
	nTileToCheck				: UINT;
	bWithBumperID				: BOOL;	
	nMoverAccessoryIdCount		: ARRAY[1..GVL.gc_nMaxNumberMovers] OF UDINT;	
	
	stStartCheck 				: ST_CheckStartConditionFeedback;
	nLimitExceeded_MoverID		: UDINT;
	bLimitExceeded_Angle 		: BOOL;
	bLimitExceeded_PositionX 	: BOOL;
	bLimitExceeded_PositionY 	: BOOL;	
	fCurrentAngleDeviation		: LREAL;
	fCurrentPositionDeviationX	: LREAL;
	fCurrentPositionDeviationY	: LREAL;	

	sTextTemp					: STRING;

	eMoverAccessoryID			: MoverAccessoryID;

	
	moverCoordComStatus			: CoordinatedMoverCommStatus;
	moverComStatus				: MoverCommunicationStatus;
	
	bMoverCommunicationProblem  : ARRAY[1..GVL.gc_nMaxNumberMovers] OF BOOL;
	bCommunicationProblem		: BOOL;
	
	nMoverToCorrect				: UDINT;
	fMoverOrientationRead		: LREAL;
	fMoverOrientationCorrect	: LREAL;
	bDoRotationCorrection		: BOOL;
	CorrectionPos				: PositionXYC;
	
	bDeterminedMoverID				: BOOL;
	bDerterminedMoverOrientation 	: BOOL;
	
	fPosX							: LREAL;
	fPosY							: LREAL;
	fPosC							: LREAL;
	
	nCommunicationRetryCounter		: UINT;
	
	nMoverToCheck					: UINT;
	
	nMoverID_ErrorCode				: DWORD;
	
	MoverType						: XPlanarMoverType;
	bMoverCanDeterminOrientation	: BOOL;
	
			// Helper
	bDone 					: BOOL;
	idx						: UDINT;
	nForCounter 			: UDINT;	
	nErrorID				: UDINT;
	bMoverError				: BOOL;	
END_VAR
VAR
	sBtn: STRING(13);
END_VAR
IF bReset THEN
	nStatePreparation := 0;
	MoverPreparation := TRUE;
END_IF


	CASE nStatePreparation OF
		
	0:  nStatePreparation := 10;
	

	10: // 1st: Check if the system is in simulation mode or not
		// Simulation > OperationMode = 1
		//     Normal > OperationMode = 0
	    operationMode := fbXPlanarSystem.ipDriver.TcIoXpu(1).GetOperationMode();	
		IF operationMode = 0 THEN
			bPowerMissing := FALSE;
			nStatePreparation := nStatePreparation + 10;
		ELSE
			nStatePreparation := 500;
		END_IF
	
		
	20: // 2nd: Check power of each tile
		(*IF NOT bPowerMissing THEN
			ipVisuMessage.SetInfoMessage('Checking tile power', 'MoverPreparation', nStatePreparation);
		ELSE
			ipVisuMessage.SetErrorMessage('Tile power missing!', 'MoverPreparation', nStatePreparation, 0);	
		END_IF*)
		
		    bPowerOK := TRUE;
		nTileToCheck := 0;
		  nTileCount := fbXPlanarSystem.ipDriver.TcIoXpu(1).GetTileCount();
		
		nStatePreparation := nStatePreparation + 1;
		
	21:
		nTileToCheck := nTileToCheck +1;
		IF nTileToCheck <= nTileCount THEN
			nStatePreparation := nStatePreparation + 1;
		ELSE
			IF bPowerOK THEN
				nStatePreparation := nStatePreparation + 9;
			ELSE
				bPowerMissing := TRUE;
				nStatePreparation := nStatePreparation - 1;
			END_IF
		END_IF
		
	22:
		nTileDcLinkVoltage := fbXPlanarSystem.ipDriver.TcIoXpu(1).TcIoTile(1,nTileToCheck).GetDcLinkVoltage(); 
		IF nTileDcLinkVoltage > 6.0 THEN
			bTilePowerOK := TRUE;
		ELSE
			bTilePowerOK := FALSE;	
		END_IF
		bPowerOK := bPowerOK AND bTilePowerOK;
		bTilePowerOverview[nTileToCheck] := bPowerOK;
		nStatePreparation := nStatePreparation - 1;
		
		
		
	30:// 3rd: Mover re-detection, in case a mover was removed inbetween
	
		// Check if a mover has been lost...
		IF fbXPlanarSystem.CheckValidMovers() THEN
			//ipVisuMessage.SetInfoMessage('Mover re-detection', 'MoverPreparation', nStatePreparation);
		
		nStatePreparation := nStatePreparation + 1;
		END_IF
	
	31:
		IF fbXPlanarSystem.P_CheckValidMovers.bDone THEN
			IF fbXPlanarSystem.P_CheckValidMovers.bMoverLost THEN
				         bDeterminedMoverID := FALSE;
				bDerterminedMoverOrientation := FALSE;
				nStatePreparation := nStatePreparation + 1;
			ELSE
				nStatePreparation := nStatePreparation + 9;
			END_IF
		END_IF
				
		bDeterminedMoverID := FALSE;
		bDerterminedMoverOrientation := FALSE;		
		
		
	32: // Starting mover re-detection
		IF fbXPlanarSystem.UtilityCheckForError(bAutoReset := TRUE) > 0 THEN
			IF fbXPlanarSystem.ipDriver.TcIoXpu(1).SetStartMoverRedetection() THEN	
				nStatePreparation := nStatePreparation +1;
			END_IF
		END_IF
	
	33: // Checking if all movers have been found on the XPlanar surface
		stMoverDetectionInfos := fbXPlanarSystem.ipDriver.TcIoXpu(1).GetMoverDetectionInfos();
		gvl.g_nMoverCount := stMoverDetectionInfos.APM4220Detected ;
		
		
		IF stMoverDetectionInfos.APM4220Detected = stMoverDetectionInfos.APM4220Expected THEN
			nStatePreparation := nStatePreparation +7;
		ELSE
			sTextTemp := 'Mover Missing!  Expected:';
			sTextTemp := CONCAT(sTextTemp, UDINT_TO_STRING(stMoverDetectionInfos.APM4220Expected));
			sTextTemp := CONCAT(sTextTemp, '  Detected:');
			sTextTemp := CONCAT(sTextTemp, UDINT_TO_STRING(stMoverDetectionInfos.APM4220Detected));
			
			//ipVisuMessage.SetErrorMessage(sTextTemp, 'MoverPreparation', nStatePreparation, 0);	
		END_IF
	
	
	 40: // 4th: Checking the position of each mover before enabeling
	 	//ipVisuMessage.SetInfoMessage('Check mover position', 'MoverPreparation', nStatePreparation);
		stMoverDetectionInfos := fbXPlanarSystem.ipDriver.TcIoXpu(1).GetMoverDetectionInfos();	 	
		gvl.g_nMoverCount := stMoverDetectionInfos.APM4220Detected ;
		
		bDone := TRUE;
		FOR idx:=1 TO GVL.g_nMoverCount DO
			stStartCheck := GVL.g_Movers[idx].std.CheckStartConditions();
			IF NOT stStartCheck.bPositionOK THEN
				bDone := FALSE;
				EXIT;
			END_IF			
		END_FOR
	
		IF bDone THEN
			nStatePreparation := nStatePreparation + 2;
		ELSE
			nStatePreparation := nStatePreparation + 1;
		END_IF
			
	 41: // Position-Check failed:
		 // Except for rotation-points between four quadrants the angle limit of the c-axis is +/- 10.0°
		 // At rotation-points the max position deviation is +/-1mm in x/y-direction  	
				nLimitExceeded_MoverID := stStartCheck.nMoverID;
				  bLimitExceeded_Angle := stStartCheck.bAngleLimitExceeded;
			  bLimitExceeded_PositionX := stStartCheck.bPositionXLimitExceeded;
			  bLimitExceeded_PositionY := stStartCheck.bPositionYLimitExceeded;	
				fCurrentAngleDeviation := stStartCheck.fCurrentAngleDeviation;
			fCurrentPositionDeviationX := stStartCheck.fCurrentPositionDeviationX;
			fCurrentPositionDeviationY := stStartCheck.fCurrentPositionDeviationY;
	
			sTextTemp := 'Position Check Failed! - Mover ';
			sTextTemp := CONCAT(sTextTemp, UDINT_TO_STRING(nLimitExceeded_MoverID));
			sTextTemp := CONCAT(sTextTemp, ' too far away from rotation point.');
			
			//ipVisuMessage.SetErrorMessage(sTextTemp, 'MoverPreparation', nStatePreparation, 0);	
			
			nStatePreparation := nStatePreparation - 1;
			
	42:		//ipVisuMessage.ClearAllMessages();
			nStatePreparation := nStatePreparation + 8;
		
		
		
	50: // 5th: Check if movers with accessory MoverID are present. If yes, do mover identification before enabeling all movers.	
		bWithBumperID := FALSE;
			
		IF fbXPlanarSystem.UtilityCheckForError(bAutoReset := TRUE) > 0 THEN
			FOR idx:=1 TO GVL.g_nMoverCount DO
				nMoverAccessoryIdCount[idx] := fbXPlanarSystem.ipDriver.TcIoXpu(1).TcIoMover(UDINT_TO_UINT(idx)).GetMoverAccessoryIdCount();
			END_FOR
			
			FOR idx:=1 TO GVL.g_nMoverCount DO
				FOR idx2:=1 TO nMoverAccessoryIdCount[idx] DO
					eMoverAccessoryID := fbXPlanarSystem.ipDriver.TcIoXpu(1).TcIoMover(UDINT_TO_UINT(idx)).GetMoverAccessoryID(UDINT_TO_INT(idx2));
					
